LIN {X -30.144,Y 21.431,Z -152.349,A 90.000,B 90.000,C 0.000} C_DIS
LIN {X -28.451,Y 21.431,Z -154.021,A 90.000,B 90.000,C 0.000} C_DIS
LIN {X -26.721,Y 21.431,Z -155.654,A 90.000,B 90.000,C 0.000} C_DIS
LIN {X -24.954,Y 21.431,Z -157.248,A 90.000,B 90.000,C 0.000} C_DIS
LIN {X -23.391,Y 21.431,Z -158.620,A 90.000,B 90.000,C 0.000} C_DIS
LIN {X -21.866,Y 21.431,Z -160.034,A 90.000,B 90.000,C 0.000} C_DIS
LIN {X -20.381,Y 21.431,Z -161.489,A 90.000,B 90.000,C 0.000} C_DIS
LIN {X -18.936,Y 21.431,Z -162.985,A 90.000,B 90.000,C 0.000} C_DIS
LIN {X -18.816,Y 21.431,Z -163.139,A 90.000,B 90.000,C 0.000} C_DIS
LIN {X -18.465,Y 21.431,Z -163.537,A 90.000,B 90.000,C 0.000} C_DIS
LIN {X -18.745,Y 21.431,Z -164.193,A 90.000,B 90.000,C 0.000} C_DIS
LIN {X -19.053,Y 21.431,Z -164.837,A 90.000,B 90.000,C 0.000} C_DIS
LIN {X -19.388,Y 21.431,Z -165.467,A 90.000,B 90.000,C 0.000} C_DIS
LIN {X -20.384,Y 21.431,Z -167.015,A 90.000,B 90.000,C 0.000} C_DIS
LIN {X -21.432,Y 21.431,Z -168.529,A 90.000,B 90.000,C 0.000} C_DIS
LIN {X -22.530,Y 21.431,Z -170.007,A 90.000,B 90.000,C 0.000} C_DIS
LIN {X -23.679,Y 21.431,Z -171.446,A 90.000,B 90.000,C 0.000} C_DIS
LIN {X -24.875,Y 21.431,Z -172.845,A 90.000,B 90.000,C 0.000} C_DIS
LIN {X -26.119,Y 21.431,Z -174.203,A 90.000,B 90.000,C 0.000} C_DIS
LIN {X -27.407,Y 21.431,Z -175.517,A 90.000,B 90.000,C 0.000} C_DIS
LIN {X -28.740,Y 21.431,Z -176.788,A 90.000,B 90.000,C 0.000} C_DIS
LIN {X -30.115,Y 21.431,Z -178.012,A 90.000,B 90.000,C 0.000} C_DIS
LIN {X -33.824,Y 21.431,Z -181.091,A 90.000,B 90.000,C 0.000} C_DIS
LIN {X -37.575,Y 21.431,Z -184.119,A 90.000,B 90.000,C 0.000} C_DIS
LIN {X -41.368,Y 21.431,Z -187.094,A 90.000,B 90.000,C 0.000} C_DIS
LIN {X -45.202,Y 21.431,Z -190.016,A 90.000,B 90.000,C 0.000} C_DIS
LIN {X -49.076,Y 21.431,Z -192.884,A 90.000,B 90.000,C 0.000} C_DIS
LIN {X -52.990,Y 21.431,Z -195.698,A 90.000,B 90.000,C 0.000} C_DIS
LIN {X -56.942,Y 21.431,Z -198.458,A 90.000,B 90.000,C 0.000} C_DIS
LIN {X -60.933,Y 21.431,Z -201.162,A 90.000,B 90.000,C 0.000} C_DIS
LIN {X -64.961,Y 21.431,Z -203.810,A 90.000,B 90.000,C 0.000} C_DIS
LIN {X -71.435,Y 21.431,Z -208.001,A 90.000,B 90.000,C 0.000} C_DIS
LIN {X -77.876,Y 21.431,Z -212.245,A 90.000,B 90.000,C 0.000} C_DIS
LIN {X -84.282,Y 21.431,Z -216.541,A 90.000,B 90.000,C 0.000} C_DIS
LIN {X -90.653,Y 21.431,Z -220.888,A 90.000,B 90.000,C 0.000} C_DIS
LIN {X -96.988,Y 21.431,Z -225.287,A 90.000,B 90.000,C 0.000} C_DIS
LIN {X -101.728,Y 21.431,Z -228.575,A 90.000,B 90.000,C 0.000} C_DIS
LIN {X -107.096,Y 21.431,Z -232.379,A 90.000,B 90.000,C 0.000} C_DIS
LIN {X -112.491,Y 21.431,Z -236.145,A 90.000,B 90.000,C 0.000} C_DIS
LIN {X -117.912,Y 21.431,Z -239.872,A 90.000,B 90.000,C 0.000} C_DIS
LIN {X -123.359,Y 21.431,Z -243.561,A 90.000,B 90.000,C 0.000} C_DIS
LIN {X -145.015,Y 21.431,Z -243.561,A 90.000,B 90.000,C 0.000} C_DIS
LIN {X -145.015,Y 21.431,Z 0.000,A 90.000,B 90.000,C 0.000} C_DIS
LIN {X -145.015,Y 33.931,Z 0.000,A 90.000,B 90.000,C 0.000} C_DIS
LIN {X -145.015,Y 46.431,Z 0.000,A 90.000,B 90.000,C 0.000} C_DIS
LIN {X -145.015,Y 55.062,Z 0.000,A 90.000,B 90.000,C 0.000} C_DIS
LIN {X 100.302,Y 55.062,Z -242.561,A 90.000,B 90.000,C 0.000} C_DIS
LIN {X 100.302,Y 39.288,Z -242.561,A 90.000,B 90.000,C 0.000} C_DIS
LIN {X 100.302,Y 26.788,Z -242.561,A 90.000,B 90.000,C 0.000} C_DIS
LIN {X 100.302,Y 14.287,Z -242.561,A 90.000,B 90.000,C 0.000} C_DIS
LIN {X 144.015,Y 14.287,Z -242.561,A 90.000,B 90.000,C 0.000} C_DIS
LIN {X 144.015,Y 14.287,Z -235.012,A 90.000,B 90.000,C 0.000} C_DIS
LIN {X 102.620,Y 14.287,Z -235.012,A 90.000,B 90.000,C 0.000} C_DIS
LIN {X 103.410,Y 14.287,Z -232.279,A 90.000,B 90.000,C 0.000} C_DIS
LIN {X 104.175,Y 14.287,Z -229.540,A 90.000,B 90.000,C 0.000} C_DIS
LIN {X 104.688,Y 14.287,Z -227.464,A 90.000,B 90.000,C 0.000} C_DIS
LIN {X 144.015,Y 14.287,Z -227.464,A 90.000,B 90.000,C 0.000} C_DIS
LIN {X 144.015,Y 14.287,Z -219.915,A 90.000,B 90.000,C 0.000} C_DIS
LIN {X 106.467,Y 14.287,Z -219.915,A 90.000,B 90.000,C 0.000} C_DIS
LIN {X 107.307,Y 14.287,Z -216.144,A 90.000,B 90.000,C 0.000} C_DIS
LIN {X 108.116,Y 14.287,Z -212.366,A 90.000,B 90.000,C 0.000} C_DIS
LIN {X 144.015,Y 14.287,Z -212.366,A 90.000,B 90.000,C 0.000} C_DIS
LIN {X 144.015,Y 14.287,Z -204.817,A 90.000,B 90.000,C 0.000} C_DIS
LIN {X 109.635,Y 14.287,Z -204.817,A 90.000,B 90.000,C 0.000} C_DIS
LIN {X 110.346,Y 14.287,Z -201.046,A 90.000,B 90.000,C 0.000} C_DIS
LIN {X 111.025,Y 14.287,Z -197.269,A 90.000,B 90.000,C 0.000} C_DIS
LIN {X 144.015,Y 14.287,Z -197.269,A 90.000,B 90.000,C 0.000} C_DIS
LIN {X 144.015,Y 14.287,Z -189.720,A 90.000,B 90.000,C 0.000} C_DIS
LIN {X 112.289,Y 14.287,Z -189.720,A 90.000,B 90.000,C 0.000} C_DIS
LIN {X 112.873,Y 14.287,Z -185.948,A 90.000,B 90.000,C 0.000} C_DIS
LIN {X 113.426,Y 14.287,Z -182.171,A 90.000,B 90.000,C 0.000} C_DIS
LIN {X 144.015,Y 14.287,Z -182.171,A 90.000,B 90.000,C 0.000} C_DIS
LIN {X 144.015,Y 14.287,Z -174.622,A 90.000,B 90.000,C 0.000} C_DIS
LIN {X 114.438,Y 14.287,Z -174.622,A 90.000,B 90.000,C 0.000} C_DIS
LIN {X 114.897,Y 14.287,Z -170.849,A 90.000,B 90.000,C 0.000} C_DIS
LIN {X 115.326,Y 14.287,Z -167.073,A 90.000,B 90.000,C 0.000} C_DIS
LIN {X 144.015,Y 14.287,Z -167.073,A 90.000,B 90.000,C 0.000} C_DIS
LIN {X 144.015,Y 14.287,Z -159.525,A 90.000,B 90.000,C 0.000} C_DIS
LIN {X 116.227,Y 14.287,Z -159.525,A 90.000,B 90.000,C 0.000} C_DIS
LIN {X 116.473,Y 14.287,Z -157.011,A 90.000,B 90.000,C 0.000} C_DIS
LIN {X 116.688,Y 14.287,Z -154.495,A 90.000,B 90.000,C 0.000} C_DIS
LIN {X 116.873,Y 14.287,Z -151.976,A 90.000,B 90.000,C 0.000} C_DIS
LIN {X 144.015,Y 14.287,Z -151.976,A 90.000,B 90.000,C 0.000} C_DIS
LIN {X 144.015,Y 14.287,Z -144.427,A 90.000,B 90.000,C 0.000} C_DIS
LIN {X 117.247,Y 14.287,Z -144.427,A 90.000,B 90.000,C 0.000} C_DIS
LIN {X 117.311,Y 14.287,Z -141.911,A 90.000,B 90.000,C 0.000} C_DIS
LIN {X 117.346,Y 14.287,Z -139.395,A 90.000,B 90.000,C 0.000} C_DIS
LIN {X 117.350,Y 14.287,Z -136.878,A 90.000,B 90.000,C 0.000} C_DIS
LIN {X 144.015,Y 14.287,Z -136.878,A 90.000,B 90.000,C 0.000} C_DIS
LIN {X 144.015,Y 14.287,Z -129.329,A 90.000,B 90.000,C 0.000} C_DIS
LIN {X 117.183,Y 14.287,Z -129.329,A 90.000,B 90.000,C 0.000} C_DIS
LIN {X 117.163,Y 14.287,Z -128.828,A 90.000,B 90.000,C 0.000} C_DIS
LIN {X 117.003,Y 14.287,Z -126.477,A 90.000,B 90.000,C 0.000} C_DIS
LIN {X 116.820,Y 14.287,Z -124.128,A 90.000,B 90.000,C 0.000} C_DIS
LIN {X 116.613,Y 14.287,Z -121.781,A 90.000,B 90.000,C 0.000} C_DIS
LIN {X 144.015,Y 14.287,Z -121.781,A 90.000,B 90.000,C 0.000} C_DIS
LIN {X 144.015,Y 14.287,Z -114.232,A 90.000,B 90.000,C 0.000} C_DIS
LIN {X 115.786,Y 14.287,Z -114.232,A 90.000,B 90.000,C 0.000} C_DIS
LIN {X 115.455,Y 14.287,Z -111.712,A 90.000,B 90.000,C 0.000} C_DIS
LIN {X 115.097,Y 14.287,Z -109.195,A 90.000,B 90.000,C 0.000} C_DIS
LIN {X 114.712,Y 14.287,Z -106.683,A 90.000,B 90.000,C 0.000} C_DIS
LIN {X 144.015,Y 14.287,Z -106.683,A 90.000,B 90.000,C 0.000} C_DIS
LIN {X 144.015,Y 14.287,Z -99.134,A 90.000,B 90.000,C 0.000} C_DIS
LIN {X 113.387,Y 14.287,Z -99.134,A 90.000,B 90.000,C 0.000} C_DIS
LIN {X 113.108,Y 14.287,Z -97.708,A 90.000,B 90.000,C 0.000} C_DIS
LIN {X 112.820,Y 14.287,Z -96.283,A 90.000,B 90.000,C 0.000} C_DIS
LIN {X 112.622,Y 14.287,Z -95.095,A 90.000,B 90.000,C 0.000} C_DIS
LIN {X 112.380,Y 14.287,Z -93.915,A 90.000,B 90.000,C 0.000} C_DIS
LIN {X 112.094,Y 14.287,Z -92.745,A 90.000,B 90.000,C 0.000} C_DIS
LIN {X 111.765,Y 14.287,Z -91.586,A 90.000,B 90.000,C 0.000} C_DIS
LIN {X 144.015,Y 14.287,Z -91.586,A 90.000,B 90.000,C 0.000} C_DIS
LIN {X 144.015,Y 14.287,Z -84.037,A 90.000,B 90.000,C 0.000} C_DIS
LIN {X 110.092,Y 14.287,Z -84.037,A 90.000,B 90.000,C 0.000} C_DIS
LIN {X 111.141,Y 14.287,Z -82.191,A 90.000,B 90.000,C 0.000} C_DIS
LIN {X 112.138,Y 14.287,Z -80.316,A 90.000,B 90.000,C 0.000} C_DIS
LIN {X 113.084,Y 14.287,Z -78.415,A 90.000,B 90.000,C 0.000} C_DIS
LIN {X 113.977,Y 14.287,Z -76.488,A 90.000,B 90.000,C 0.000} C_DIS
LIN {X 144.015,Y 14.287,Z -76.488,A 90.000,B 90.000,C 0.000} C_DIS
LIN {X 144.015,Y 14.287,Z -68.939,A 90.000,B 90.000,C 0.000} C_DIS
LIN {X 116.890,Y 14.287,Z -68.939,A 90.000,B 90.000,C 0.000} C_DIS
LIN {X 117.231,Y 14.287,Z -67.869,A 90.000,B 90.000,C 0.000} C_DIS
LIN {X 117.556,Y 14.287,Z -66.794,A 90.000,B 90.000,C 0.000} C_DIS
LIN {X 118.300,Y 14.287,Z -64.088,A 90.000,B 90.000,C 0.000} C_DIS
LIN {X 119.069,Y 14.287,Z -61.390,A 90.000,B 90.000,C 0.000} C_DIS
LIN {X 144.015,Y 14.287,Z -61.390,A 90.000,B 90.000,C 0.000} C_DIS
LIN {X 144.015,Y 14.287,Z -53.842,A 90.000,B 90.000,C 0.000} C_DIS
LIN {X 122.274,Y 14.287,Z -53.842,A 90.000,B 90.000,C 0.000} C_DIS
LIN {X 122.630,Y 14.287,Z -53.139,A 90.000,B 90.000,C 0.000} C_DIS
LIN {X 122.993,Y 14.287,Z -52.439,A 90.000,B 90.000,C 0.000} C_DIS
LIN {X 123.486,Y 14.287,Z -51.468,A 90.000,B 90.000,C 0.000} C_DIS
LIN {X 123.926,Y 14.287,Z -50.472,A 90.000,B 90.000,C 0.000} C_DIS
LIN {X 124.312,Y 14.287,Z -49.453,A 90.000,B 90.000,C 0.000} C_DIS
LIN {X 124.641,Y 14.287,Z -48.415,A 90.000,B 90.000,C 0.000} C_DIS
LIN {X 124.915,Y 14.287,Z -47.360,A 90.000,B 90.000,C 0.000} C_DIS
LIN {X 125.131,Y 14.287,Z -46.293,A 90.000,B 90.000,C 0.000} C_DIS
LIN {X 144.015,Y 14.287,Z -46.293,A 90.000,B 90.000,C 0.000} C_DIS
LIN {X 144.015,Y 14.287,Z -38.744,A 90.000,B 90.000,C 0.000} C_DIS
LIN {X 125.030,Y 14.287,Z -38.744,A 90.000,B 90.000,C 0.000} C_DIS
LIN {X 124.784,Y 14.287,Z -37.789,A 90.000,B 90.000,C 0.000} C_DIS
LIN {X 124.472,Y 14.287,Z -36.853,A 90.000,B 90.000,C 0.000} C_DIS
LIN {X 124.097,Y 14.287,Z -35.940,A 90.000,B 90.000,C 0.000} C_DIS
LIN {X 123.660,Y 14.287,Z -35.056,A 90.000,B 90.000,C 0.000} C_DIS
LIN {X 123.164,Y 14.287,Z -34.204,A 90.000,B 90.000,C 0.000} C_DIS
LIN {X 122.609,Y 14.287,Z -33.388,A 90.000,B 90.000,C 0.000} C_DIS
LIN {X 122.000,Y 14.287,Z -32.612,A 90.000,B 90.000,C 0.000} C_DIS
LIN {X 121.339,Y 14.287,Z -31.880,A 90.000,B 90.000,C 0.000} C_DIS
LIN {X 120.629,Y 14.287,Z -31.195,A 90.000,B 90.000,C 0.000} C_DIS
LIN {X 144.015,Y 14.287,Z -31.195,A 90.000,B 90.000,C 0.000} C_DIS
LIN {X 144.015,Y 14.287,Z -23.646,A 90.000,B 90.000,C 0.000} C_DIS
LIN {X 5.340,Y 14.287,Z -23.646,A 90.000,B 90.000,C 0.000} C_DIS
LIN {X 2.315,Y 14.287,Z -23.147,A 90.000,B 90.000,C 0.000} C_DIS
LIN {X -0.703,Y 14.287,Z -22.607,A 90.000,B 90.000,C 0.000} C_DIS
LIN {X -3.714,Y 14.287,Z -22.027,A 90.000,B 90.000,C 0.000} C_DIS
LIN {X -6.716,Y 14.287,Z -21.406,A 90.000,B 90.000,C 0.000} C_DIS
LIN {X -9.710,Y 14.287,Z -20.745,A 90.000,B 90.000,C 0.000} C_DIS
LIN {X -13.667,Y 14.287,Z -19.813,A 90.000,B 90.000,C 0.000} C_DIS
LIN {X -17.634,Y 14.287,Z -18.928,A 90.000,B 90.000,C 0.000} C_DIS
LIN {X -21.612,Y 14.287,Z -18.088,A 90.000,B 90.000,C 0.000} C_DIS
LIN {X -25.599,Y 14.287,Z -17.295,A 90.000,B 90.000,C 0.000} C_DIS
LIN {X -27.541,Y 14.287,Z -16.862,A 90.000,B 90.000,C 0.000} C_DIS
LIN {X -29.491,Y 14.287,Z -16.463,A 90.000,B 90.000,C 0.000} C_DIS
LIN {X -31.447,Y 14.287,Z -16.098,A 90.000,B 90.000,C 0.000} C_DIS
LIN {X 144.015,Y 14.287,Z -16.098,A 90.000,B 90.000,C 0.000} C_DIS
LIN {X 144.015,Y 14.287,Z -8.549,A 90.000,B 90.000,C 0.000} C_DIS
LIN {X -67.014,Y 14.287,Z -8.549,A 90.000,B 90.000,C 0.000} C_DIS
LIN {X -68.321,Y 14.287,Z -7.964,A 90.000,B 90.000,C 0.000} C_DIS
LIN {X -69.464,Y 14.287,Z -7.415,A 90.000,B 90.000,C 0.000} C_DIS
LIN {X -70.635,Y 14.287,Z -6.927,A 90.000,B 90.000,C 0.000} C_DIS
LIN {X -71.829,Y 14.287,Z -6.502,A 90.000,B 90.000,C 0.000} C_DIS
LIN {X -73.045,Y 14.287,Z -6.142,A 90.000,B 90.000,C 0.000} C_DIS
LIN {X -74.279,Y 14.287,Z -5.847,A 90.000,B 90.000,C 0.000} C_DIS
LIN {X -75.526,Y 14.287,Z -5.618,A 90.000,B 90.000,C 0.000} C_DIS
LIN {X -76.784,Y 14.287,Z -5.456,A 90.000,B 90.000,C 0.000} C_DIS
LIN {X -78.048,Y 14.287,Z -5.361,A 90.000,B 90.000,C 0.000} C_DIS
LIN {X -79.316,Y 14.287,Z -5.334,A 90.000,B 90.000,C 0.000} C_DIS
LIN {X -80.584,Y 14.287,Z -5.375,A 90.000,B 90.000,C 0.000} C_DIS
LIN {X -81.847,Y 14.287,Z -5.483,A 90.000,B 90.000,C 0.000} C_DIS
LIN {X -83.103,Y 14.287,Z -5.658,A 90.000,B 90.000,C 0.000} C_DIS
LIN {X -84.348,Y 14.287,Z -5.899,A 90.000,B 90.000,C 0.000} C_DIS
LIN {X -85.303,Y 14.287,Z -6.093,A 90.000,B 90.000,C 0.000} C_DIS
LIN {X -86.243,Y 14.287,Z -6.351,A 90.000,B 90.000,C 0.000} C_DIS
LIN {X -87.163,Y 14.287,Z -6.671,A 90.000,B 90.000,C 0.000} C_DIS
LIN {X -88.060,Y 14.287,Z -7.052,A 90.000,B 90.000,C 0.000} C_DIS
LIN {X -88.929,Y 14.287,Z -7.492,A 90.000,B 90.000,C 0.000} C_DIS
LIN {X -89.767,Y 14.287,Z -7.990,A 90.000,B 90.000,C 0.000} C_DIS
LIN {X -90.843,Y 14.287,Z -8.053,A 90.000,B 90.000,C 0.000} C_DIS
LIN {X -91.915,Y 14.287,Z -8.167,A 90.000,B 90.000,C 0.000} C_DIS
LIN {X -92.981,Y 14.287,Z -8.332,A 90.000,B 90.000,C 0.000} C_DIS
LIN {X -94.037,Y 14.287,Z -8.549,A 90.000,B 90.000,C 0.000} C_DIS
LIN {X -144.015,Y 14.287,Z -8.549,A 90.000,B 90.000,C 0.000} C_DIS
LIN {X -144.015,Y 14.287,Z -16.098,A 90.000,B 90.000,C 0.000} C_DIS
LIN {X -106.655,Y 14.287,Z -16.098,A 90.000,B 90.000,C 0.000} C_DIS
LIN {X -107.024,Y 14.287,Z -16.531,A 90.000,B 90.000,C 0.000} C_DIS
LIN {X -107.373,Y 14.287,Z -16.981,A 90.000,B 90.000,C 0.000} C_DIS
LIN {X -108.462,Y 14.287,Z -17.322,A 90.000,B 90.000,C 0.000} C_DIS
LIN {X -109.531,Y 14.287,Z -17.720,A 90.000,B 90.000,C 0.000} C_DIS
LIN {X -110.578,Y 14.287,Z -18.174,A 90.000,B 90.000,C 0.000} C_DIS
LIN {X -111.598,Y 14.287,Z -18.684,A 90.000,B 90.000,C 0.000} C_DIS
LIN {X -112.591,Y 14.287,Z -19.246,A 90.000,B 90.000,C 0.000} C_DIS
LIN {X -113.552,Y 14.287,Z -19.861,A 90.000,B 90.000,C 0.000} C_DIS
LIN {X -114.479,Y 14.287,Z -20.526,A 90.000,B 90.000,C 0.000} C_DIS
LIN {X -115.370,Y 14.287,Z -21.239,A 90.000,B 90.000,C 0.000} C_DIS
LIN {X -116.222,Y 14.287,Z -21.998,A 90.000,B 90.000,C 0.000} C_DIS
LIN {X -117.032,Y 14.287,Z -22.801,A 90.000,B 90.000,C 0.000} C_DIS
LIN {X -117.799,Y 14.287,Z -23.646,A 90.000,B 90.000,C 0.000} C_DIS
LIN {X -144.015,Y 14.287,Z -23.646,A 90.000,B 90.000,C 0.000} C_DIS
LIN {X -144.015,Y 14.287,Z -31.195,A 90.000,B 90.000,C 0.000} C_DIS
LIN {X -122.817,Y 14.287,Z -31.195,A 90.000,B 90.000,C 0.000} C_DIS
LIN {X -123.177,Y 14.287,Z -32.233,A 90.000,B 90.000,C 0.000} C_DIS
LIN {X -123.472,Y 14.287,Z -33.291,A 90.000,B 90.000,C 0.000} C_DIS
LIN {X -123.701,Y 14.287,Z -34.366,A 90.000,B 90.000,C 0.000} C_DIS
LIN {X -123.861,Y 14.287,Z -35.453,A 90.000,B 90.000,C 0.000} C_DIS
LIN {X -123.954,Y 14.287,Z -36.548,A 90.000,B 90.000,C 0.000} C_DIS
LIN {X -123.979,Y 14.287,Z -37.646,A 90.000,B 90.000,C 0.000} C_DIS
LIN {X -123.934,Y 14.287,Z -38.744,A 90.000,B 90.000,C 0.000} C_DIS
LIN {X -144.015,Y 14.287,Z -38.744,A 90.000,B 90.000,C 0.000} C_DIS
LIN {X -144.015,Y 14.287,Z -46.293,A 90.000,B 90.000,C 0.000} C_DIS
LIN {X -123.207,Y 14.287,Z -46.293,A 90.000,B 90.000,C 0.000} C_DIS
LIN {X -123.190,Y 14.287,Z -47.313,A 90.000,B 90.000,C 0.000} C_DIS
LIN {X -123.108,Y 14.287,Z -48.329,A 90.000,B 90.000,C 0.000} C_DIS
LIN {X -122.962,Y 14.287,Z -49.339,A 90.000,B 90.000,C 0.000} C_DIS
LIN {X -122.752,Y 14.287,Z -50.337,A 90.000,B 90.000,C 0.000} C_DIS
LIN {X -122.479,Y 14.287,Z -51.320,A 90.000,B 90.000,C 0.000} C_DIS
LIN {X -122.144,Y 14.287,Z -52.283,A 90.000,B 90.000,C 0.000} C_DIS
LIN {X -121.748,Y 14.287,Z -53.223,A 90.000,B 90.000,C 0.000} C_DIS
LIN {X -121.595,Y 14.287,Z -53.842,A 90.000,B 90.000,C 0.000} C_DIS
LIN {X -144.015,Y 14.287,Z -53.842,A 90.000,B 90.000,C 0.000} C_DIS
LIN {X -144.015,Y 14.287,Z -61.390,A 90.000,B 90.000,C 0.000} C_DIS
LIN {X -119.537,Y 14.287,Z -61.390,A 90.000,B 90.000,C 0.000} C_DIS
LIN {X -119.056,Y 14.287,Z -62.708,A 90.000,B 90.000,C 0.000} C_DIS
LIN {X -118.522,Y 14.287,Z -64.005,A 90.000,B 90.000,C 0.000} C_DIS
LIN {X -117.934,Y 14.287,Z -65.279,A 90.000,B 90.000,C 0.000} C_DIS
LIN {X -117.295,Y 14.287,Z -66.527,A 90.000,B 90.000,C 0.000} C_DIS
LIN {X -116.604,Y 14.287,Z -67.748,A 90.000,B 90.000,C 0.000} C_DIS
LIN {X -115.863,Y 14.287,Z -68.939,A 90.000,B 90.000,C 0.000} C_DIS
LIN {X -144.015,Y 14.287,Z -68.939,A 90.000,B 90.000,C 0.000} C_DIS
LIN {X -144.015,Y 14.287,Z -76.488,A 90.000,B 90.000,C 0.000} C_DIS
LIN {X -109.288,Y 14.287,Z -76.488,A 90.000,B 90.000,C 0.000} C_DIS
LIN {X -108.521,Y 14.287,Z -77.148,A 90.000,B 90.000,C 0.000} C_DIS
LIN {X -107.719,Y 14.287,Z -77.766,A 90.000,B 90.000,C 0.000} C_DIS
LIN {X -106.886,Y 14.287,Z -78.340,A 90.000,B 90.000,C 0.000} C_DIS
LIN {X -106.023,Y 14.287,Z -78.868,A 90.000,B 90.000,C 0.000} C_DIS
LIN {X -105.133,Y 14.287,Z -79.350,A 90.000,B 90.000,C 0.000} C_DIS
LIN {X -104.218,Y 14.287,Z -79.783,A 90.000,B 90.000,C 0.000} C_DIS
LIN {X -104.128,Y 14.287,Z -79.831,A 90.000,B 90.000,C 0.000} C_DIS
LIN {X -103.286,Y 14.287,Z -80.260,A 90.000,B 90.000,C 0.000} C_DIS
LIN {X -102.420,Y 14.287,Z -80.639,A 90.000,B 90.000,C 0.000} C_DIS
LIN {X -101.534,Y 14.287,Z -80.966,A 90.000,B 90.000,C 0.000} C_DIS
LIN {X -100.630,Y 14.287,Z -81.241,A 90.000,B 90.000,C 0.000} C_DIS
LIN {X -99.711,Y 14.287,Z -81.461,A 90.000,B 90.000,C 0.000} C_DIS
LIN {X -98.781,Y 14.287,Z -81.628,A 90.000,B 90.000,C 0.000} C_DIS
LIN {X -98.628,Y 14.287,Z -81.664,A 90.000,B 90.000,C 0.000} C_DIS
LIN {X -96.905,Y 14.287,Z -81.904,A 90.000,B 90.000,C 0.000} C_DIS
LIN {X -95.177,Y 14.287,Z -82.109,A 90.000,B 90.000,C 0.000} C_DIS
LIN {X -93.445,Y 14.287,Z -82.279,A 90.000,B 90.000,C 0.000} C_DIS
LIN {X -93.383,Y 14.287,Z -82.289,A 90.000,B 90.000,C 0.000} C_DIS
LIN {X -92.938,Y 14.287,Z -82.457,A 90.000,B 90.000,C 0.000} C_DIS
LIN {X -92.507,Y 14.287,Z -82.659,A 90.000,B 90.000,C 0.000} C_DIS
LIN {X -92.093,Y 14.287,Z -82.893,A 90.000,B 90.000,C 0.000} C_DIS
LIN {X -91.698,Y 14.287,Z -83.159,A 90.000,B 90.000,C 0.000} C_DIS
LIN {X -91.216,Y 14.287,Z -83.601,A 90.000,B 90.000,C 0.000} C_DIS
LIN {X -90.729,Y 14.287,Z -84.037,A 90.000,B 90.000,C 0.000} C_DIS
LIN {X -144.015,Y 14.287,Z -84.037,A 90.000,B 90.000,C 0.000} C_DIS
LIN {X -144.015,Y 14.287,Z -91.586,A 90.000,B 90.000,C 0.000} C_DIS
LIN {X -80.184,Y 14.287,Z -91.586,A 90.000,B 90.000,C 0.000} C_DIS
LIN {X -78.153,Y 14.287,Z -92.888,A 90.000,B 90.000,C 0.000} C_DIS
LIN {X -76.910,Y 14.287,Z -93.660,A 90.000,B 90.000,C 0.000} C_DIS
LIN {X -75.693,Y 14.287,Z -94.474,A 90.000,B 90.000,C 0.000} C_DIS
LIN {X -74.505,Y 14.287,Z -95.329,A 90.000,B 90.000,C 0.000} C_DIS
LIN {X -73.346,Y 14.287,Z -96.223,A 90.000,B 90.000,C 0.000} C_DIS
LIN {X -72.219,Y 14.287,Z -97.156,A 90.000,B 90.000,C 0.000} C_DIS
LIN {X -71.123,Y 14.287,Z -98.127,A 90.000,B 90.000,C 0.000} C_DIS
LIN {X -70.061,Y 14.287,Z -99.134,A 90.000,B 90.000,C 0.000} C_DIS
LIN {X -144.015,Y 14.287,Z -99.134,A 90.000,B 90.000,C 0.000} C_DIS
LIN {X -144.015,Y 14.287,Z -106.683,A 90.000,B 90.000,C 0.000} C_DIS
LIN {X -63.845,Y 14.287,Z -106.683,A 90.000,B 90.000,C 0.000} C_DIS
LIN {X -61.945,Y 14.287,Z -109.223,A 90.000,B 90.000,C 0.000} C_DIS
LIN {X -60.014,Y 14.287,Z -111.739,A 90.000,B 90.000,C 0.000} C_DIS
LIN {X -58.052,Y 14.287,Z -114.232,A 90.000,B 90.000,C 0.000} C_DIS
LIN {X -144.015,Y 14.287,Z -114.232,A 90.000,B 90.000,C 0.000} C_DIS
LIN {X -144.015,Y 14.287,Z -121.781,A 90.000,B 90.000,C 0.000} C_DIS
LIN {X -51.816,Y 14.287,Z -121.781,A 90.000,B 90.000,C 0.000} C_DIS
LIN {X -50.808,Y 14.287,Z -123.147,A 90.000,B 90.000,C 0.000} C_DIS
LIN {X -49.834,Y 14.287,Z -124.538,A 90.000,B 90.000,C 0.000} C_DIS
LIN {X -49.055,Y 14.287,Z -126.117,A 90.000,B 90.000,C 0.000} C_DIS
LIN {X -48.313,Y 14.287,Z -127.715,A 90.000,B 90.000,C 0.000} C_DIS
LIN {X -47.609,Y 14.287,Z -129.329,A 90.000,B 90.000,C 0.000} C_DIS
LIN {X -144.015,Y 14.287,Z -129.329,A 90.000,B 90.000,C 0.000} C_DIS
LIN {X -144.015,Y 14.287,Z -136.878,A 90.000,B 90.000,C 0.000} C_DIS
LIN {X -44.292,Y 14.287,Z -136.878,A 90.000,B 90.000,C 0.000} C_DIS
LIN {X -43.485,Y 14.287,Z -138.431,A 90.000,B 90.000,C 0.000} C_DIS
LIN {X -42.639,Y 14.287,Z -139.963,A 90.000,B 90.000,C 0.000} C_DIS
LIN {X -41.756,Y 14.287,Z -141.473,A 90.000,B 90.000,C 0.000} C_DIS
LIN {X -40.836,Y 14.287,Z -142.962,A 90.000,B 90.000,C 0.000} C_DIS
LIN {X -39.879,Y 14.287,Z -144.427,A 90.000,B 90.000,C 0.000} C_DIS
LIN {X -144.015,Y 14.287,Z -144.427,A 90.000,B 90.000,C 0.000} C_DIS
LIN {X -144.015,Y 14.287,Z -151.976,A 90.000,B 90.000,C 0.000} C_DIS
LIN {X -33.972,Y 14.287,Z -151.976,A 90.000,B 90.000,C 0.000} C_DIS
LIN {X -31.573,Y 14.287,Z -154.527,A 90.000,B 90.000,C 0.000} C_DIS
LIN {X -29.138,Y 14.287,Z -157.044,A 90.000,B 90.000,C 0.000} C_DIS
LIN {X -26.667,Y 14.287,Z -159.525,A 90.000,B 90.000,C 0.000} C_DIS
LIN {X -144.015,Y 14.287,Z -159.525,A 90.000,B 90.000,C 0.000} C_DIS
LIN {X -144.015,Y 14.287,Z -167.073,A 90.000,B 90.000,C 0.000} C_DIS
LIN {X -26.448,Y 14.287,Z -167.073,A 90.000,B 90.000,C 0.000} C_DIS
LIN {X -27.323,Y 14.287,Z -168.257,A 90.000,B 90.000,C 0.000} C_DIS
LIN {X -28.242,Y 14.287,Z -169.409,A 90.000,B 90.000,C 0.000} C_DIS
LIN {X -29.201,Y 14.287,Z -170.526,A 90.000,B 90.000,C 0.000} C_DIS
LIN {X -30.201,Y 14.287,Z -171.607,A 90.000,B 90.000,C 0.000} C_DIS
LIN {X -31.239,Y 14.287,Z -172.651,A 90.000,B 90.000,C 0.000} C_DIS
LIN {X -32.315,Y 14.287,Z -173.657,A 90.000,B 90.000,C 0.000} C_DIS
LIN {X -33.427,Y 14.287,Z -174.622,A 90.000,B 90.000,C 0.000} C_DIS
LIN {X -144.015,Y 14.287,Z -174.622,A 90.000,B 90.000,C 0.000} C_DIS
LIN {X -144.015,Y 14.287,Z -182.171,A 90.000,B 90.000,C 0.000} C_DIS
LIN {X -43.393,Y 14.287,Z -182.171,A 90.000,B 90.000,C 0.000} C_DIS
LIN {X -46.143,Y 14.287,Z -184.116,A 90.000,B 90.000,C 0.000} C_DIS
LIN {X -48.919,Y 14.287,Z -186.023,A 90.000,B 90.000,C 0.000} C_DIS
LIN {X -51.722,Y 14.287,Z -187.891,A 90.000,B 90.000,C 0.000} C_DIS
LIN {X -54.550,Y 14.287,Z -189.720,A 90.000,B 90.000,C 0.000} C_DIS
LIN {X -144.015,Y 14.287,Z -189.720,A 90.000,B 90.000,C 0.000} C_DIS
LIN {X -144.015,Y 14.287,Z -197.269,A 90.000,B 90.000,C 0.000} C_DIS
LIN {X -66.947,Y 14.287,Z -197.269,A 90.000,B 90.000,C 0.000} C_DIS
LIN {X -71.176,Y 14.287,Z -199.763,A 90.000,B 90.000,C 0.000} C_DIS
LIN {X -75.391,Y 14.287,Z -202.279,A 90.000,B 90.000,C 0.000} C_DIS
LIN {X -79.594,Y 14.287,Z -204.817,A 90.000,B 90.000,C 0.000} C_DIS
LIN {X -144.015,Y 14.287,Z -204.817,A 90.000,B 90.000,C 0.000} C_DIS
LIN {X -144.015,Y 14.287,Z -212.366,A 90.000,B 90.000,C 0.000} C_DIS
LIN {X -91.801,Y 14.287,Z -212.366,A 90.000,B 90.000,C 0.000} C_DIS
LIN {X -95.747,Y 14.287,Z -214.862,A 90.000,B 90.000,C 0.000} C_DIS
LIN {X -99.680,Y 14.287,Z -217.379,A 90.000,B 90.000,C 0.000} C_DIS
LIN {X -103.600,Y 14.287,Z -219.915,A 90.000,B 90.000,C 0.000} C_DIS
LIN {X -144.015,Y 14.287,Z -219.915,A 90.000,B 90.000,C 0.000} C_DIS
LIN {X -144.015,Y 14.287,Z -227.464,A 90.000,B 90.000,C 0.000} C_DIS
LIN {X -115.053,Y 14.287,Z -227.464,A 90.000,B 90.000,C 0.000} C_DIS
LIN {X -122.337,Y 14.287,Z -232.351,A 90.000,B 90.000,C 0.000} C_DIS
LIN {X -126.258,Y 14.287,Z -235.012,A 90.000,B 90.000,C 0.000} C_DIS
LIN {X -144.015,Y 14.287,Z -235.012,A 90.000,B 90.000,C 0.000} C_DIS
LIN {X -144.015,Y 14.287,Z -242.561,A 90.000,B 90.000,C 0.000} C_DIS
LIN {X -137.094,Y 14.287,Z -242.561,A 90.000,B 90.000,C 0.000} C_DIS
LIN {X -144.015,Y 14.287,Z -1.000,A 90.000,B 90.000,C 0.000} C_DIS
LIN {X 144.015,Y 14.287,Z -1.000,A 90.000,B 90.000,C 0.000} C_DIS
LIN {X 98.307,Y 14.287,Z -31.195,A 90.000,B 90.000,C 0.000} C_DIS
LIN {X 45.099,Y 14.287,Z -31.195,A 90.000,B 90.000,C 0.000} C_DIS
LIN {X 47.546,Y 14.287,Z -32.059,A 90.000,B 90.000,C 0.000} C_DIS
LIN {X 49.978,Y 14.287,Z -32.965,A 90.000,B 90.000,C 0.000} C_DIS
LIN {X 52.394,Y 14.287,Z -33.911,A 90.000,B 90.000,C 0.000} C_DIS
LIN {X 54.085,Y 14.287,Z -34.773,A 90.000,B 90.000,C 0.000} C_DIS
LIN {X 55.748,Y 14.287,Z -35.689,A 90.000,B 90.000,C 0.000} C_DIS
LIN {X 57.382,Y 14.287,Z -36.656,A 90.000,B 90.000,C 0.000} C_DIS
LIN {X 58.983,Y 14.287,Z -37.675,A 90.000,B 90.000,C 0.000} C_DIS
LIN {X 60.552,Y 14.287,Z -38.744,A 90.000,B 90.000,C 0.000} C_DIS
LIN {X 85.592,Y 14.287,Z -38.744,A 90.000,B 90.000,C 0.000} C_DIS
LIN {X 84.450,Y 14.287,Z -39.711,A 90.000,B 90.000,C 0.000} C_DIS
LIN {X 83.338,Y 14.287,Z -40.714,A 90.000,B 90.000,C 0.000} C_DIS
LIN {X 82.260,Y 14.287,Z -41.752,A 90.000,B 90.000,C 0.000} C_DIS
LIN {X 81.214,Y 14.287,Z -42.823,A 90.000,B 90.000,C 0.000} C_DIS
LIN {X 80.413,Y 14.287,Z -43.639,A 90.000,B 90.000,C 0.000} C_DIS
LIN {X 79.650,Y 14.287,Z -44.490,A 90.000,B 90.000,C 0.000} C_DIS
LIN {X 78.927,Y 14.287,Z -45.375,A 90.000,B 90.000,C 0.000} C_DIS
LIN {X 78.245,Y 14.287,Z -46.293,A 90.000,B 90.000,C 0.000} C_DIS
LIN {X 73.847,Y 14.287,Z -46.293,A 90.000,B 90.000,C 0.000} C_DIS
LIN {X 77.376,Y 14.287,Z -49.619,A 90.000,B 90.000,C 0.000} C_DIS
LIN {X 75.302,Y 14.287,Z -48.325,A 90.000,B 90.000,C 0.000} C_DIS
LIN {X 73.202,Y 14.287,Z -47.074,A 90.000,B 90.000,C 0.000} C_DIS
LIN {X 71.075,Y 14.287,Z -45.869,A 90.000,B 90.000,C 0.000} C_DIS
LIN {X 68.924,Y 14.287,Z -44.709,A 90.000,B 90.000,C 0.000} C_DIS
LIN {X 66.748,Y 14.287,Z -43.594,A 90.000,B 90.000,C 0.000} C_DIS
LIN {X 64.550,Y 14.287,Z -42.525,A 90.000,B 90.000,C 0.000} C_DIS
LIN {X 63.559,Y 14.287,Z -42.002,A 90.000,B 90.000,C 0.000} C_DIS
LIN {X 62.561,Y 14.287,Z -41.493,A 90.000,B 90.000,C 0.000} C_DIS
LIN {X 61.141,Y 14.287,Z -40.405,A 90.000,B 90.000,C 0.000} C_DIS
LIN {X 59.688,Y 14.287,Z -39.360,A 90.000,B 90.000,C 0.000} C_DIS
LIN {X 58.204,Y 14.287,Z -38.361,A 90.000,B 90.000,C 0.000} C_DIS
LIN {X 56.691,Y 14.287,Z -37.406,A 90.000,B 90.000,C 0.000} C_DIS
LIN {X 55.149,Y 14.287,Z -36.498,A 90.000,B 90.000,C 0.000} C_DIS
LIN {X 53.581,Y 14.287,Z -35.638,A 90.000,B 90.000,C 0.000} C_DIS
LIN {X 51.987,Y 14.287,Z -34.825,A 90.000,B 90.000,C 0.000} C_DIS
LIN {X 49.331,Y 14.287,Z -33.789,A 90.000,B 90.000,C 0.000} C_DIS
LIN {X 46.657,Y 14.287,Z -32.802,A 90.000,B 90.000,C 0.000} C_DIS
LIN {X 43.964,Y 14.287,Z -31.865,A 90.000,B 90.000,C 0.000} C_DIS
LIN {X 41.255,Y 14.287,Z -30.978,A 90.000,B 90.000,C 0.000} C_DIS
LIN {X 38.529,Y 14.287,Z -30.142,A 90.000,B 90.000,C 0.000} C_DIS
LIN {X 35.789,Y 14.287,Z -29.356,A 90.000,B 90.000,C 0.000} C_DIS
LIN {X 33.956,Y 14.287,Z -28.833,A 90.000,B 90.000,C 0.000} C_DIS
LIN {X 32.105,Y 14.287,Z -28.373,A 90.000,B 90.000,C 0.000} C_DIS
LIN {X 30.240,Y 14.287,Z -27.976,A 90.000,B 90.000,C 0.000} C_DIS
LIN {X 28.363,Y 14.287,Z -27.644,A 90.000,B 90.000,C 0.000} C_DIS
LIN {X 26.475,Y 14.287,Z -27.375,A 90.000,B 90.000,C 0.000} C_DIS
LIN {X 24.580,Y 14.287,Z -27.172,A 90.000,B 90.000,C 0.000} C_DIS
LIN {X 22.678,Y 14.287,Z -27.034,A 90.000,B 90.000,C 0.000} C_DIS
LIN {X 21.240,Y 14.287,Z -27.123,A 90.000,B 90.000,C 0.000} C_DIS
LIN {X 19.800,Y 14.287,Z -27.159,A 90.000,B 90.000,C 0.000} C_DIS
LIN {X 18.359,Y 14.287,Z -27.141,A 90.000,B 90.000,C 0.000} C_DIS
LIN {X 16.920,Y 14.287,Z -27.069,A 90.000,B 90.000,C 0.000} C_DIS
LIN {X 13.486,Y 14.287,Z -26.291,A 90.000,B 90.000,C 0.000} C_DIS
LIN {X 10.044,Y 14.287,Z -25.553,A 90.000,B 90.000,C 0.000} C_DIS
LIN {X 6.594,Y 14.287,Z -24.852,A 90.000,B 90.000,C 0.000} C_DIS
LIN {X 3.270,Y 14.287,Z -24.323,A 90.000,B 90.000,C 0.000} C_DIS
LIN {X -0.047,Y 14.287,Z -23.745,A 90.000,B 90.000,C 0.000} C_DIS
LIN {X -3.354,Y 14.287,Z -23.118,A 90.000,B 90.000,C 0.000} C_DIS
LIN {X -6.651,Y 14.287,Z -22.442,A 90.000,B 90.000,C 0.000} C_DIS
LIN {X -9.939,Y 14.287,Z -21.719,A 90.000,B 90.000,C 0.000} C_DIS
LIN {X -13.891,Y 14.287,Z -20.789,A 90.000,B 90.000,C 0.000} C_DIS
LIN {X -17.853,Y 14.287,Z -19.904,A 90.000,B 90.000,C 0.000} C_DIS
LIN {X -21.825,Y 14.287,Z -19.066,A 90.000,B 90.000,C 0.000} C_DIS
LIN {X -25.807,Y 14.287,Z -18.274,A 90.000,B 90.000,C 0.000} C_DIS
LIN {X -27.926,Y 14.287,Z -17.803,A 90.000,B 90.000,C 0.000} C_DIS
LIN {X -30.054,Y 14.287,Z -17.373,A 90.000,B 90.000,C 0.000} C_DIS
LIN {X -32.189,Y 14.287,Z -16.983,A 90.000,B 90.000,C 0.000} C_DIS
LIN {X -34.331,Y 14.287,Z -16.634,A 90.000,B 90.000,C 0.000} C_DIS
LIN {X -36.480,Y 14.287,Z -16.326,A 90.000,B 90.000,C 0.000} C_DIS
LIN {X -39.917,Y 14.287,Z -15.920,A 90.000,B 90.000,C 0.000} C_DIS
LIN {X -43.352,Y 14.287,Z -15.497,A 90.000,B 90.000,C 0.000} C_DIS
LIN {X -48.382,Y 14.287,Z -14.794,A 90.000,B 90.000,C 0.000} C_DIS
LIN {X -53.417,Y 14.287,Z -14.125,A 90.000,B 90.000,C 0.000} C_DIS
LIN {X -54.230,Y 14.287,Z -14.089,A 90.000,B 90.000,C 0.000} C_DIS
LIN {X -55.040,Y 14.287,Z -14.011,A 90.000,B 90.000,C 0.000} C_DIS
LIN {X -55.845,Y 14.287,Z -13.891,A 90.000,B 90.000,C 0.000} C_DIS
LIN {X -56.643,Y 14.287,Z -13.730,A 90.000,B 90.000,C 0.000} C_DIS
LIN {X -57.431,Y 14.287,Z -13.528,A 90.000,B 90.000,C 0.000} C_DIS
LIN {X -60.292,Y 14.287,Z -12.436,A 90.000,B 90.000,C 0.000} C_DIS
LIN {X -63.134,Y 14.287,Z -11.294,A 90.000,B 90.000,C 0.000} C_DIS
LIN {X -65.956,Y 14.287,Z -10.104,A 90.000,B 90.000,C 0.000} C_DIS
LIN {X -68.756,Y 14.287,Z -8.864,A 90.000,B 90.000,C 0.000} C_DIS
LIN {X -69.854,Y 14.287,Z -8.335,A 90.000,B 90.000,C 0.000} C_DIS
LIN {X -70.978,Y 14.287,Z -7.865,A 90.000,B 90.000,C 0.000} C_DIS
LIN {X -72.126,Y 14.287,Z -7.457,A 90.000,B 90.000,C 0.000} C_DIS
LIN {X -73.295,Y 14.287,Z -7.110,A 90.000,B 90.000,C 0.000} C_DIS
LIN {X -74.480,Y 14.287,Z -6.826,A 90.000,B 90.000,C 0.000} C_DIS
LIN {X -75.679,Y 14.287,Z -6.606,A 90.000,B 90.000,C 0.000} C_DIS
LIN {X -76.887,Y 14.287,Z -6.450,A 90.000,B 90.000,C 0.000} C_DIS
LIN {X -78.103,Y 14.287,Z -6.359,A 90.000,B 90.000,C 0.000} C_DIS
LIN {X -79.321,Y 14.287,Z -6.334,A 90.000,B 90.000,C 0.000} C_DIS
LIN {X -80.539,Y 14.287,Z -6.373,A 90.000,B 90.000,C 0.000} C_DIS
LIN {X -81.753,Y 14.287,Z -6.478,A 90.000,B 90.000,C 0.000} C_DIS
LIN {X -82.960,Y 14.287,Z -6.647,A 90.000,B 90.000,C 0.000} C_DIS
LIN {X -84.156,Y 14.287,Z -6.881,A 90.000,B 90.000,C 0.000} C_DIS
LIN {X -84.961,Y 14.287,Z -7.040,A 90.000,B 90.000,C 0.000} C_DIS
LIN {X -85.755,Y 14.287,Z -7.248,A 90.000,B 90.000,C 0.000} C_DIS
LIN {X -86.535,Y 14.287,Z -7.504,A 90.000,B 90.000,C 0.000} C_DIS
LIN {X -87.298,Y 14.287,Z -7.806,A 90.000,B 90.000,C 0.000} C_DIS
LIN {X -88.041,Y 14.287,Z -8.154,A 90.000,B 90.000,C 0.000} C_DIS
LIN {X -88.761,Y 14.287,Z -8.547,A 90.000,B 90.000,C 0.000} C_DIS
LIN {X -89.457,Y 14.287,Z -8.982,A 90.000,B 90.000,C 0.000} C_DIS
LIN {X -90.658,Y 14.287,Z -9.041,A 90.000,B 90.000,C 0.000} C_DIS
LIN {X -91.853,Y 14.287,Z -9.168,A 90.000,B 90.000,C 0.000} C_DIS
LIN {X -93.040,Y 14.287,Z -9.361,A 90.000,B 90.000,C 0.000} C_DIS
LIN {X -94.214,Y 14.287,Z -9.619,A 90.000,B 90.000,C 0.000} C_DIS
LIN {X -95.371,Y 14.287,Z -9.943,A 90.000,B 90.000,C 0.000} C_DIS
LIN {X -96.509,Y 14.287,Z -10.331,A 90.000,B 90.000,C 0.000} C_DIS
LIN {X -96.645,Y 14.287,Z -10.387,A 90.000,B 90.000,C 0.000} C_DIS
LIN {X -97.481,Y 14.287,Z -10.765,A 90.000,B 90.000,C 0.000} C_DIS
LIN {X -98.293,Y 14.287,Z -11.190,A 90.000,B 90.000,C 0.000} C_DIS
LIN {X -99.080,Y 14.287,Z -11.662,A 90.000,B 90.000,C 0.000} C_DIS
LIN {X -99.839,Y 14.287,Z -12.177,A 90.000,B 90.000,C 0.000} C_DIS
LIN {X -100.563,Y 14.287,Z -12.778,A 90.000,B 90.000,C 0.000} C_DIS
LIN {X -101.300,Y 14.287,Z -13.364,A 90.000,B 90.000,C 0.000} C_DIS
LIN {X -102.049,Y 14.287,Z -13.933,A 90.000,B 90.000,C 0.000} C_DIS
LIN {X -102.843,Y 14.287,Z -14.328,A 90.000,B 90.000,C 0.000} C_DIS
LIN {X -103.604,Y 14.287,Z -14.782,A 90.000,B 90.000,C 0.000} C_DIS
LIN {X -104.328,Y 14.287,Z -15.295,A 90.000,B 90.000,C 0.000} C_DIS
LIN {X -105.010,Y 14.287,Z -15.861,A 90.000,B 90.000,C 0.000} C_DIS
LIN {X -105.647,Y 14.287,Z -16.478,A 90.000,B 90.000,C 0.000} C_DIS
LIN {X -106.234,Y 14.287,Z -17.143,A 90.000,B 90.000,C 0.000} C_DIS
LIN {X -106.767,Y 14.287,Z -17.851,A 90.000,B 90.000,C 0.000} C_DIS
LIN {X -107.879,Y 14.287,Z -18.181,A 90.000,B 90.000,C 0.000} C_DIS
LIN {X -108.971,Y 14.287,Z -18.573,A 90.000,B 90.000,C 0.000} C_DIS
LIN {X -110.039,Y 14.287,Z -19.027,A 90.000,B 90.000,C 0.000} C_DIS
LIN {X -111.079,Y 14.287,Z -19.540,A 90.000,B 90.000,C 0.000} C_DIS
LIN {X -112.089,Y 14.287,Z -20.111,A 90.000,B 90.000,C 0.000} C_DIS
LIN {X -113.065,Y 14.287,Z -20.739,A 90.000,B 90.000,C 0.000} C_DIS
LIN {X -114.004,Y 14.287,Z -21.420,A 90.000,B 90.000,C 0.000} C_DIS
LIN {X -114.902,Y 14.287,Z -22.154,A 90.000,B 90.000,C 0.000} C_DIS
LIN {X -115.758,Y 14.287,Z -22.937,A 90.000,B 90.000,C 0.000} C_DIS
LIN {X -116.568,Y 14.287,Z -23.768,A 90.000,B 90.000,C 0.000} C_DIS
LIN {X -117.330,Y 14.287,Z -24.643,A 90.000,B 90.000,C 0.000} C_DIS
LIN {X -117.877,Y 14.287,Z -25.450,A 90.000,B 90.000,C 0.000} C_DIS
LIN {X -118.467,Y 14.287,Z -26.225,A 90.000,B 90.000,C 0.000} C_DIS
LIN {X -119.099,Y 14.287,Z -26.967,A 90.000,B 90.000,C 0.000} C_DIS
LIN {X -119.770,Y 14.287,Z -27.674,A 90.000,B 90.000,C 0.000} C_DIS
LIN {X -120.392,Y 14.287,Z -28.586,A 90.000,B 90.000,C 0.000} C_DIS
LIN {X -120.953,Y 14.287,Z -29.537,A 90.000,B 90.000,C 0.000} C_DIS
LIN {X -121.449,Y 14.287,Z -30.524,A 90.000,B 90.000,C 0.000} C_DIS
LIN {X -121.878,Y 14.287,Z -31.541,A 90.000,B 90.000,C 0.000} C_DIS
LIN {X -122.239,Y 14.287,Z -32.584,A 90.000,B 90.000,C 0.000} C_DIS
LIN {X -122.529,Y 14.287,Z -33.649,A 90.000,B 90.000,C 0.000} C_DIS
LIN {X -122.749,Y 14.287,Z -34.732,A 90.000,B 90.000,C 0.000} C_DIS
LIN {X -122.895,Y 14.287,Z -35.826,A 90.000,B 90.000,C 0.000} C_DIS
LIN {X -122.969,Y 14.287,Z -36.927,A 90.000,B 90.000,C 0.000} C_DIS
LIN {X -122.970,Y 14.287,Z -38.031,A 90.000,B 90.000,C 0.000} C_DIS
LIN {X -122.897,Y 14.287,Z -39.133,A 90.000,B 90.000,C 0.000} C_DIS
LIN {X -122.751,Y 14.287,Z -40.228,A 90.000,B 90.000,C 0.000} C_DIS
LIN {X -122.532,Y 14.287,Z -41.310,A 90.000,B 90.000,C 0.000} C_DIS
LIN {X -122.243,Y 14.287,Z -42.375,A 90.000,B 90.000,C 0.000} C_DIS
LIN {X -121.883,Y 14.287,Z -43.419,A 90.000,B 90.000,C 0.000} C_DIS
LIN {X -122.053,Y 14.287,Z -44.374,A 90.000,B 90.000,C 0.000} C_DIS
LIN {X -122.161,Y 14.287,Z -45.338,A 90.000,B 90.000,C 0.000} C_DIS
LIN {X -122.207,Y 14.287,Z -46.307,A 90.000,B 90.000,C 0.000} C_DIS
LIN {X -122.191,Y 14.287,Z -47.277,A 90.000,B 90.000,C 0.000} C_DIS
LIN {X -122.111,Y 14.287,Z -48.244,A 90.000,B 90.000,C 0.000} C_DIS
LIN {X -121.970,Y 14.287,Z -49.204,A 90.000,B 90.000,C 0.000} C_DIS
LIN {X -121.767,Y 14.287,Z -50.153,A 90.000,B 90.000,C 0.000} C_DIS
LIN {X -121.504,Y 14.287,Z -51.086,A 90.000,B 90.000,C 0.000} C_DIS
LIN {X -121.181,Y 14.287,Z -52.001,A 90.000,B 90.000,C 0.000} C_DIS
LIN {X -120.799,Y 14.287,Z -52.893,A 90.000,B 90.000,C 0.000} C_DIS
LIN {X -120.485,Y 14.287,Z -54.139,A 90.000,B 90.000,C 0.000} C_DIS
LIN {X -120.143,Y 14.287,Z -55.377,A 90.000,B 90.000,C 0.000} C_DIS
LIN {X -119.772,Y 14.287,Z -56.607,A 90.000,B 90.000,C 0.000} C_DIS
LIN {X -119.454,Y 14.287,Z -58.085,A 90.000,B 90.000,C 0.000} C_DIS
LIN {X -119.069,Y 14.287,Z -59.546,A 90.000,B 90.000,C 0.000} C_DIS
LIN {X -118.617,Y 14.287,Z -60.988,A 90.000,B 90.000,C 0.000} C_DIS
LIN {X -118.100,Y 14.287,Z -62.408,A 90.000,B 90.000,C 0.000} C_DIS
LIN {X -117.518,Y 14.287,Z -63.803,A 90.000,B 90.000,C 0.000} C_DIS
LIN {X -116.873,Y 14.287,Z -65.170,A 90.000,B 90.000,C 0.000} C_DIS
LIN {X -116.165,Y 14.287,Z -66.506,A 90.000,B 90.000,C 0.000} C_DIS
LIN {X -115.398,Y 14.287,Z -67.808,A 90.000,B 90.000,C 0.000} C_DIS
LIN {X -114.571,Y 14.287,Z -69.073,A 90.000,B 90.000,C 0.000} C_DIS
LIN {X -113.687,Y 14.287,Z -70.299,A 90.000,B 90.000,C 0.000} C_DIS
LIN {X -112.748,Y 14.287,Z -71.483,A 90.000,B 90.000,C 0.000} C_DIS
LIN {X -111.756,Y 14.287,Z -72.623,A 90.000,B 90.000,C 0.000} C_DIS
LIN {X -110.712,Y 14.287,Z -73.717,A 90.000,B 90.000,C 0.000} C_DIS
LIN {X -109.620,Y 14.287,Z -74.761,A 90.000,B 90.000,C 0.000} C_DIS
LIN {X -108.894,Y 14.287,Z -75.489,A 90.000,B 90.000,C 0.000} C_DIS
LIN {X -108.128,Y 14.287,Z -76.175,A 90.000,B 90.000,C 0.000} C_DIS
LIN {X -107.324,Y 14.287,Z -76.815,A 90.000,B 90.000,C 0.000} C_DIS
LIN {X -106.484,Y 14.287,Z -77.407,A 90.000,B 90.000,C 0.000} C_DIS
LIN {X -105.611,Y 14.287,Z -77.951,A 90.000,B 90.000,C 0.000} C_DIS
LIN {X -104.709,Y 14.287,Z -78.444,A 90.000,B 90.000,C 0.000} C_DIS
LIN {X -103.780,Y 14.287,Z -78.884,A 90.000,B 90.000,C 0.000} C_DIS
LIN {X -103.652,Y 14.287,Z -78.952,A 90.000,B 90.000,C 0.000} C_DIS
LIN {X -102.856,Y 14.287,Z -79.358,A 90.000,B 90.000,C 0.000} C_DIS
LIN {X -102.037,Y 14.287,Z -79.716,A 90.000,B 90.000,C 0.000} C_DIS
LIN {X -101.198,Y 14.287,Z -80.024,A 90.000,B 90.000,C 0.000} C_DIS
LIN {X -100.343,Y 14.287,Z -80.283,A 90.000,B 90.000,C 0.000} C_DIS
LIN {X -99.473,Y 14.287,Z -80.490,A 90.000,B 90.000,C 0.000} C_DIS
LIN {X -98.593,Y 14.287,Z -80.645,A 90.000,B 90.000,C 0.000} C_DIS
LIN {X -98.439,Y 14.287,Z -80.681,A 90.000,B 90.000,C 0.000} C_DIS
LIN {X -96.737,Y 14.287,Z -80.917,A 90.000,B 90.000,C 0.000} C_DIS
LIN {X -95.031,Y 14.287,Z -81.118,A 90.000,B 90.000,C 0.000} C_DIS
LIN {X -93.321,Y 14.287,Z -81.286,A 90.000,B 90.000,C 0.000} C_DIS
LIN {X -93.146,Y 14.287,Z -81.314,A 90.000,B 90.000,C 0.000} C_DIS
LIN {X -92.593,Y 14.287,Z -81.517,A 90.000,B 90.000,C 0.000} C_DIS
LIN {X -92.058,Y 14.287,Z -81.764,A 90.000,B 90.000,C 0.000} C_DIS
LIN {X -91.545,Y 14.287,Z -82.055,A 90.000,B 90.000,C 0.000} C_DIS
LIN {X -91.059,Y 14.287,Z -82.388,A 90.000,B 90.000,C 0.000} C_DIS
LIN {X -89.751,Y 14.287,Z -83.565,A 90.000,B 90.000,C 0.000} C_DIS
LIN {X -88.408,Y 14.287,Z -84.701,A 90.000,B 90.000,C 0.000} C_DIS
LIN {X -87.030,Y 14.287,Z -85.794,A 90.000,B 90.000,C 0.000} C_DIS
LIN {X -85.619,Y 14.287,Z -86.845,A 90.000,B 90.000,C 0.000} C_DIS
LIN {X -84.177,Y 14.287,Z -87.853,A 90.000,B 90.000,C 0.000} C_DIS
LIN {X -82.704,Y 14.287,Z -88.815,A 90.000,B 90.000,C 0.000} C_DIS
LIN {X -80.158,Y 14.287,Z -90.417,A 90.000,B 90.000,C 0.000} C_DIS
LIN {X -77.625,Y 14.287,Z -92.039,A 90.000,B 90.000,C 0.000} C_DIS
LIN {X -76.194,Y 14.287,Z -92.933,A 90.000,B 90.000,C 0.000} C_DIS
LIN {X -74.799,Y 14.287,Z -93.880,A 90.000,B 90.000,C 0.000} C_DIS
LIN {X -73.441,Y 14.287,Z -94.880,A 90.000,B 90.000,C 0.000} C_DIS
LIN {X -72.121,Y 14.287,Z -95.931,A 90.000,B 90.000,C 0.000} C_DIS
LIN {X -70.843,Y 14.287,Z -97.032,A 90.000,B 90.000,C 0.000} C_DIS
LIN {X -69.608,Y 14.287,Z -98.180,A 90.000,B 90.000,C 0.000} C_DIS
LIN {X -68.417,Y 14.287,Z -99.375,A 90.000,B 90.000,C 0.000} C_DIS
LIN {X -67.273,Y 14.287,Z -100.614,A 90.000,B 90.000,C 0.000} C_DIS
LIN {X -66.177,Y 14.287,Z -101.897,A 90.000,B 90.000,C 0.000} C_DIS
LIN {X -65.130,Y 14.287,Z -103.219,A 90.000,B 90.000,C 0.000} C_DIS
LIN {X -63.219,Y 14.287,Z -105.846,A 90.000,B 90.000,C 0.000} C_DIS
LIN {X -61.276,Y 14.287,Z -108.449,A 90.000,B 90.000,C 0.000} C_DIS
LIN {X -59.300,Y 14.287,Z -111.027,A 90.000,B 90.000,C 0.000} C_DIS
LIN {X -57.292,Y 14.287,Z -113.581,A 90.000,B 90.000,C 0.000} C_DIS
LIN {X -55.252,Y 14.287,Z -116.109,A 90.000,B 90.000,C 0.000} C_DIS
LIN {X -53.905,Y 14.287,Z -117.618,A 90.000,B 90.000,C 0.000} C_DIS
LIN {X -52.602,Y 14.287,Z -119.166,A 90.000,B 90.000,C 0.000} C_DIS
LIN {X -51.345,Y 14.287,Z -120.751,A 90.000,B 90.000,C 0.000} C_DIS
LIN {X -50.134,Y 14.287,Z -122.372,A 90.000,B 90.000,C 0.000} C_DIS
LIN {X -48.971,Y 14.287,Z -124.028,A 90.000,B 90.000,C 0.000} C_DIS
LIN {X -48.160,Y 14.287,Z -125.670,A 90.000,B 90.000,C 0.000} C_DIS
LIN {X -47.389,Y 14.287,Z -127.330,A 90.000,B 90.000,C 0.000} C_DIS
LIN {X -46.658,Y 14.287,Z -129.010,A 90.000,B 90.000,C 0.000} C_DIS
LIN {X -45.969,Y 14.287,Z -130.706,A 90.000,B 90.000,C 0.000} C_DIS
LIN {X -45.181,Y 14.287,Z -132.612,A 90.000,B 90.000,C 0.000} C_DIS
LIN {X -44.337,Y 14.287,Z -134.494,A 90.000,B 90.000,C 0.000} C_DIS
LIN {X -43.438,Y 14.287,Z -136.350,A 90.000,B 90.000,C 0.000} C_DIS
LIN {X -42.485,Y 14.287,Z -138.179,A 90.000,B 90.000,C 0.000} C_DIS
LIN {X -41.477,Y 14.287,Z -139.979,A 90.000,B 90.000,C 0.000} C_DIS
LIN {X -40.417,Y 14.287,Z -141.748,A 90.000,B 90.000,C 0.000} C_DIS
LIN {X -39.305,Y 14.287,Z -143.485,A 90.000,B 90.000,C 0.000} C_DIS
LIN {X -38.142,Y 14.287,Z -145.188,A 90.000,B 90.000,C 0.000} C_DIS
LIN {X -36.929,Y 14.287,Z -146.856,A 90.000,B 90.000,C 0.000} C_DIS
LIN {X -35.667,Y 14.287,Z -148.488,A 90.000,B 90.000,C 0.000} C_DIS
LIN {X -34.357,Y 14.287,Z -150.081,A 90.000,B 90.000,C 0.000} C_DIS
LIN {X -32.177,Y 14.287,Z -152.435,A 90.000,B 90.000,C 0.000} C_DIS
LIN {X -29.965,Y 14.287,Z -154.761,A 90.000,B 90.000,C 0.000} C_DIS
LIN {X -27.722,Y 14.287,Z -157.056,A 90.000,B 90.000,C 0.000} C_DIS
LIN {X -25.449,Y 14.287,Z -159.321,A 90.000,B 90.000,C 0.000} C_DIS
LIN {X -24.833,Y 14.287,Z -159.908,A 90.000,B 90.000,C 0.000} C_DIS
LIN {X -24.254,Y 14.287,Z -160.532,A 90.000,B 90.000,C 0.000} C_DIS
LIN {X -23.714,Y 14.287,Z -161.190,A 90.000,B 90.000,C 0.000} C_DIS
LIN {X -23.215,Y 14.287,Z -161.879,A 90.000,B 90.000,C 0.000} C_DIS
LIN {X -22.758,Y 14.287,Z -162.597,A 90.000,B 90.000,C 0.000} C_DIS
LIN {X -23.115,Y 14.287,Z -163.460,A 90.000,B 90.000,C 0.000} C_DIS
LIN {X -23.519,Y 14.287,Z -164.302,A 90.000,B 90.000,C 0.000} C_DIS
LIN {X -23.968,Y 14.287,Z -165.121,A 90.000,B 90.000,C 0.000} C_DIS
LIN {X -24.780,Y 14.287,Z -166.407,A 90.000,B 90.000,C 0.000} C_DIS
LIN {X -25.640,Y 14.287,Z -167.662,A 90.000,B 90.000,C 0.000} C_DIS
LIN {X -26.544,Y 14.287,Z -168.885,A 90.000,B 90.000,C 0.000} C_DIS
LIN {X -27.494,Y 14.287,Z -170.073,A 90.000,B 90.000,C 0.000} C_DIS
LIN {X -28.486,Y 14.287,Z -171.226,A 90.000,B 90.000,C 0.000} C_DIS
LIN {X -29.520,Y 14.287,Z -172.342,A 90.000,B 90.000,C 0.000} C_DIS
LIN {X -30.594,Y 14.287,Z -173.419,A 90.000,B 90.000,C 0.000} C_DIS
LIN {X -31.707,Y 14.287,Z -174.455,A 90.000,B 90.000,C 0.000} C_DIS
LIN {X -32.858,Y 14.287,Z -175.450,A 90.000,B 90.000,C 0.000} C_DIS
LIN {X -35.875,Y 14.287,Z -177.819,A 90.000,B 90.000,C 0.000} C_DIS
LIN {X -38.929,Y 14.287,Z -180.140,A 90.000,B 90.000,C 0.000} C_DIS
LIN {X -42.019,Y 14.287,Z -182.413,A 90.000,B 90.000,C 0.000} C_DIS
LIN {X -45.144,Y 14.287,Z -184.637,A 90.000,B 90.000,C 0.000} C_DIS
LIN {X -48.303,Y 14.287,Z -186.813,A 90.000,B 90.000,C 0.000} C_DIS
LIN {X -51.496,Y 14.287,Z -188.938,A 90.000,B 90.000,C 0.000} C_DIS
LIN {X -54.722,Y 14.287,Z -191.013,A 90.000,B 90.000,C 0.000} C_DIS
LIN {X -57.980,Y 14.287,Z -193.038,A 90.000,B 90.000,C 0.000} C_DIS
LIN {X -61.453,Y 14.287,Z -195.127,A 90.000,B 90.000,C 0.000} C_DIS
LIN {X -64.912,Y 14.287,Z -197.237,A 90.000,B 90.000,C 0.000} C_DIS
LIN {X -70.964,Y 14.287,Z -200.799,A 90.000,B 90.000,C 0.000} C_DIS
LIN {X -76.988,Y 14.287,Z -204.408,A 90.000,B 90.000,C 0.000} C_DIS
LIN {X -82.985,Y 14.287,Z -208.062,A 90.000,B 90.000,C 0.000} C_DIS
LIN {X -88.954,Y 14.287,Z -211.761,A 90.000,B 90.000,C 0.000} C_DIS
LIN {X -94.895,Y 14.287,Z -215.506,A 90.000,B 90.000,C 0.000} C_DIS
LIN {X -100.807,Y 14.287,Z -219.296,A 90.000,B 90.000,C 0.000} C_DIS
LIN {X -106.690,Y 14.287,Z -223.130,A 90.000,B 90.000,C 0.000} C_DIS
LIN {X -114.380,Y 14.287,Z -228.216,A 90.000,B 90.000,C 0.000} C_DIS
LIN {X -121.778,Y 14.287,Z -233.180,A 90.000,B 90.000,C 0.000} C_DIS
LIN {X -128.845,Y 14.287,Z -237.978,A 90.000,B 90.000,C 0.000} C_DIS
LIN {X -135.503,Y 14.287,Z -242.529,A 90.000,B 90.000,C 0.000} C_DIS
LIN {X -136.644,Y 14.287,Z -243.489,A 90.000,B 90.000,C 0.000} C_DIS
LIN {X -136.709,Y 14.287,Z -243.561,A 90.000,B 90.000,C 0.000} C_DIS
LIN {X -145.015,Y 14.287,Z -243.561,A 90.000,B 90.000,C 0.000} C_DIS
LIN {X -145.015,Y 14.287,Z 0.000,A 90.000,B 90.000,C 0.000} C_DIS
LIN {X 145.015,Y 14.287,Z 0.000,A 90.000,B 90.000,C 0.000} C_DIS
LIN {X 145.015,Y 14.287,Z -243.561,A 90.000,B 90.000,C 0.000} C_DIS
LIN {X 98.929,Y 14.287,Z -243.561,A 90.000,B 90.000,C 0.000} C_DIS
LIN {X 100.061,Y 14.287,Z -240.011,A 90.000,B 90.000,C 0.000} C_DIS
LIN {X 101.151,Y 14.287,Z -236.449,A 90.000,B 90.000,C 0.000} C_DIS
LIN {X 102.200,Y 14.287,Z -232.874,A 90.000,B 90.000,C 0.000} C_DIS
LIN {X 103.208,Y 14.287,Z -229.287,A 90.000,B 90.000,C 0.000} C_DIS
LIN {X 104.581,Y 14.287,Z -223.630,A 90.000,B 90.000,C 0.000} C_DIS
LIN {X 105.883,Y 14.287,Z -217.956,A 90.000,B 90.000,C 0.000} C_DIS
LIN {X 107.115,Y 14.287,Z -212.267,A 90.000,B 90.000,C 0.000} C_DIS
LIN {X 108.276,Y 14.287,Z -206.563,A 90.000,B 90.000,C 0.000} C_DIS
LIN {X 109.366,Y 14.287,Z -200.845,A 90.000,B 90.000,C 0.000} C_DIS
LIN {X 110.385,Y 14.287,Z -195.113,A 90.000,B 90.000,C 0.000} C_DIS
LIN {X 111.332,Y 14.287,Z -189.370,A 90.000,B 90.000,C 0.000} C_DIS
LIN {X 112.208,Y 14.287,Z -183.615,A 90.000,B 90.000,C 0.000} C_DIS
LIN {X 113.012,Y 14.287,Z -177.850,A 90.000,B 90.000,C 0.000} C_DIS
LIN {X 113.745,Y 14.287,Z -172.075,A 90.000,B 90.000,C 0.000} C_DIS
LIN {X 114.405,Y 14.287,Z -166.291,A 90.000,B 90.000,C 0.000} C_DIS
LIN {X 114.881,Y 14.287,Z -162.571,A 90.000,B 90.000,C 0.000} C_DIS
LIN {X 115.291,Y 14.287,Z -158.844,A 90.000,B 90.000,C 0.000} C_DIS
LIN {X 115.635,Y 14.287,Z -155.109,A 90.000,B 90.000,C 0.000} C_DIS
LIN {X 115.911,Y 14.287,Z -151.369,A 90.000,B 90.000,C 0.000} C_DIS
LIN {X 116.121,Y 14.287,Z -147.625,A 90.000,B 90.000,C 0.000} C_DIS
LIN {X 116.263,Y 14.287,Z -143.877,A 90.000,B 90.000,C 0.000} C_DIS
LIN {X 116.339,Y 14.287,Z -140.128,A 90.000,B 90.000,C 0.000} C_DIS
LIN {X 116.348,Y 14.287,Z -136.378,A 90.000,B 90.000,C 0.000} C_DIS
LIN {X 116.289,Y 14.287,Z -132.628,A 90.000,B 90.000,C 0.000} C_DIS
LIN {X 116.164,Y 14.287,Z -128.880,A 90.000,B 90.000,C 0.000} C_DIS
LIN {X 115.907,Y 14.287,Z -125.252,A 90.000,B 90.000,C 0.000} C_DIS
LIN {X 115.594,Y 14.287,Z -121.628,A 90.000,B 90.000,C 0.000} C_DIS
LIN {X 115.225,Y 14.287,Z -118.009,A 90.000,B 90.000,C 0.000} C_DIS
LIN {X 114.799,Y 14.287,Z -114.397,A 90.000,B 90.000,C 0.000} C_DIS
LIN {X 114.318,Y 14.287,Z -110.791,A 90.000,B 90.000,C 0.000} C_DIS
LIN {X 113.781,Y 14.287,Z -107.194,A 90.000,B 90.000,C 0.000} C_DIS
LIN {X 113.188,Y 14.287,Z -103.605,A 90.000,B 90.000,C 0.000} C_DIS
LIN {X 112.539,Y 14.287,Z -100.026,A 90.000,B 90.000,C 0.000} C_DIS
LIN {X 111.835,Y 14.287,Z -96.457,A 90.000,B 90.000,C 0.000} C_DIS
LIN {X 111.589,Y 14.287,Z -95.017,A 90.000,B 90.000,C 0.000} C_DIS
LIN {X 111.277,Y 14.287,Z -93.591,A 90.000,B 90.000,C 0.000} C_DIS
LIN {X 110.899,Y 14.287,Z -92.180,A 90.000,B 90.000,C 0.000} C_DIS
LIN {X 110.455,Y 14.287,Z -90.788,A 90.000,B 90.000,C 0.000} C_DIS
LIN {X 109.948,Y 14.287,Z -89.419,A 90.000,B 90.000,C 0.000} C_DIS
LIN {X 109.378,Y 14.287,Z -88.074,A 90.000,B 90.000,C 0.000} C_DIS
LIN {X 108.745,Y 14.287,Z -86.758,A 90.000,B 90.000,C 0.000} C_DIS
LIN {X 108.053,Y 14.287,Z -85.472,A 90.000,B 90.000,C 0.000} C_DIS
LIN {X 109.254,Y 14.287,Z -83.491,A 90.000,B 90.000,C 0.000} C_DIS
LIN {X 110.393,Y 14.287,Z -81.474,A 90.000,B 90.000,C 0.000} C_DIS
LIN {X 111.472,Y 14.287,Z -79.424,A 90.000,B 90.000,C 0.000} C_DIS
LIN {X 112.487,Y 14.287,Z -77.342,A 90.000,B 90.000,C 0.000} C_DIS
LIN {X 113.439,Y 14.287,Z -75.230,A 90.000,B 90.000,C 0.000} C_DIS
LIN {X 114.327,Y 14.287,Z -73.090,A 90.000,B 90.000,C 0.000} C_DIS
LIN {X 115.149,Y 14.287,Z -70.924,A 90.000,B 90.000,C 0.000} C_DIS
LIN {X 115.905,Y 14.287,Z -68.735,A 90.000,B 90.000,C 0.000} C_DIS
LIN {X 116.594,Y 14.287,Z -66.523,A 90.000,B 90.000,C 0.000} C_DIS
LIN {X 117.391,Y 14.287,Z -63.629,A 90.000,B 90.000,C 0.000} C_DIS
LIN {X 118.216,Y 14.287,Z -60.743,A 90.000,B 90.000,C 0.000} C_DIS
LIN {X 118.900,Y 14.287,Z -58.947,A 90.000,B 90.000,C 0.000} C_DIS
LIN {X 119.632,Y 14.287,Z -57.170,A 90.000,B 90.000,C 0.000} C_DIS
LIN {X 120.411,Y 14.287,Z -55.413,A 90.000,B 90.000,C 0.000} C_DIS
LIN {X 121.238,Y 14.287,Z -53.679,A 90.000,B 90.000,C 0.000} C_DIS
LIN {X 122.112,Y 14.287,Z -51.967,A 90.000,B 90.000,C 0.000} C_DIS
LIN {X 122.620,Y 14.287,Z -50.961,A 90.000,B 90.000,C 0.000} C_DIS
LIN {X 123.069,Y 14.287,Z -49.926,A 90.000,B 90.000,C 0.000} C_DIS
LIN {X 123.455,Y 14.287,Z -48.867,A 90.000,B 90.000,C 0.000} C_DIS
LIN {X 123.778,Y 14.287,Z -47.788,A 90.000,B 90.000,C 0.000} C_DIS
LIN {X 124.038,Y 14.287,Z -46.690,A 90.000,B 90.000,C 0.000} C_DIS
LIN {X 124.232,Y 14.287,Z -45.580,A 90.000,B 90.000,C 0.000} C_DIS
LIN {X 124.360,Y 14.287,Z -44.460,A 90.000,B 90.000,C 0.000} C_DIS
LIN {X 124.422,Y 14.287,Z -43.334,A 90.000,B 90.000,C 0.000} C_DIS
LIN {X 124.417,Y 14.287,Z -42.207,A 90.000,B 90.000,C 0.000} C_DIS
LIN {X 124.347,Y 14.287,Z -41.082,A 90.000,B 90.000,C 0.000} C_DIS
LIN {X 124.254,Y 14.287,Z -40.095,A 90.000,B 90.000,C 0.000} C_DIS
LIN {X 124.088,Y 14.287,Z -39.117,A 90.000,B 90.000,C 0.000} C_DIS
LIN {X 123.849,Y 14.287,Z -38.155,A 90.000,B 90.000,C 0.000} C_DIS
LIN {X 123.540,Y 14.287,Z -37.213,A 90.000,B 90.000,C 0.000} C_DIS
LIN {X 123.161,Y 14.287,Z -36.296,A 90.000,B 90.000,C 0.000} C_DIS
LIN {X 122.715,Y 14.287,Z -35.411,A 90.000,B 90.000,C 0.000} C_DIS
LIN {X 122.205,Y 14.287,Z -34.561,A 90.000,B 90.000,C 0.000} C_DIS
LIN {X 121.633,Y 14.287,Z -33.751,A 90.000,B 90.000,C 0.000} C_DIS
LIN {X 121.002,Y 14.287,Z -32.986,A 90.000,B 90.000,C 0.000} C_DIS
LIN {X 120.316,Y 14.287,Z -32.270,A 90.000,B 90.000,C 0.000} C_DIS
LIN {X 119.578,Y 14.287,Z -31.607,A 90.000,B 90.000,C 0.000} C_DIS
LIN {X 118.794,Y 14.287,Z -31.001,A 90.000,B 90.000,C 0.000} C_DIS
LIN {X 117.966,Y 14.287,Z -30.455,A 90.000,B 90.000,C 0.000} C_DIS
LIN {X 117.834,Y 14.287,Z -30.373,A 90.000,B 90.000,C 0.000} C_DIS
LIN {X 117.055,Y 14.287,Z -29.942,A 90.000,B 90.000,C 0.000} C_DIS
LIN {X 116.250,Y 14.287,Z -29.561,A 90.000,B 90.000,C 0.000} C_DIS
LIN {X 115.424,Y 14.287,Z -29.230,A 90.000,B 90.000,C 0.000} C_DIS
LIN {X 114.578,Y 14.287,Z -28.952,A 90.000,B 90.000,C 0.000} C_DIS
LIN {X 114.396,Y 14.287,Z -28.894,A 90.000,B 90.000,C 0.000} C_DIS
LIN {X 113.507,Y 14.287,Z -28.671,A 90.000,B 90.000,C 0.000} C_DIS
LIN {X 112.605,Y 14.287,Z -28.507,A 90.000,B 90.000,C 0.000} C_DIS
LIN {X 111.695,Y 14.287,Z -28.401,A 90.000,B 90.000,C 0.000} C_DIS
LIN {X 110.779,Y 14.287,Z -28.354,A 90.000,B 90.000,C 0.000} C_DIS
LIN {X 109.863,Y 14.287,Z -28.367,A 90.000,B 90.000,C 0.000} C_DIS
LIN {X 108.949,Y 14.287,Z -28.439,A 90.000,B 90.000,C 0.000} C_DIS
LIN {X 108.042,Y 14.287,Z -28.571,A 90.000,B 90.000,C 0.000} C_DIS
LIN {X 107.145,Y 14.287,Z -28.761,A 90.000,B 90.000,C 0.000} C_DIS
LIN {X 105.009,Y 14.287,Z -29.519,A 90.000,B 90.000,C 0.000} C_DIS
LIN {X 102.893,Y 14.287,Z -30.330,A 90.000,B 90.000,C 0.000} C_DIS
LIN {X 100.797,Y 14.287,Z -31.192,A 90.000,B 90.000,C 0.000} C_DIS
LIN {X 98.723,Y 14.287,Z -32.105,A 90.000,B 90.000,C 0.000} C_DIS
LIN {X 96.671,Y 14.287,Z -33.068,A 90.000,B 90.000,C 0.000} C_DIS
LIN {X 95.024,Y 14.287,Z -33.842,A 90.000,B 90.000,C 0.000} C_DIS
LIN {X 93.410,Y 14.287,Z -34.680,A 90.000,B 90.000,C 0.000} C_DIS
LIN {X 91.829,Y 14.287,Z -35.581,A 90.000,B 90.000,C 0.000} C_DIS
LIN {X 90.286,Y 14.287,Z -36.544,A 90.000,B 90.000,C 0.000} C_DIS
LIN {X 88.781,Y 14.287,Z -37.567,A 90.000,B 90.000,C 0.000} C_DIS
LIN {X 87.318,Y 14.287,Z -38.649,A 90.000,B 90.000,C 0.000} C_DIS
LIN {X 85.899,Y 14.287,Z -39.787,A 90.000,B 90.000,C 0.000} C_DIS
LIN {X 84.526,Y 14.287,Z -40.981,A 90.000,B 90.000,C 0.000} C_DIS
LIN {X 83.201,Y 14.287,Z -42.228,A 90.000,B 90.000,C 0.000} C_DIS
LIN {X 81.926,Y 14.287,Z -43.526,A 90.000,B 90.000,C 0.000} C_DIS
LIN {X 81.037,Y 14.287,Z -44.437,A 90.000,B 90.000,C 0.000} C_DIS
LIN {X 80.197,Y 14.287,Z -45.393,A 90.000,B 90.000,C 0.000} C_DIS
LIN {X 79.409,Y 14.287,Z -46.392,A 90.000,B 90.000,C 0.000} C_DIS
LIN {X 78.675,Y 14.287,Z -47.431,A 90.000,B 90.000,C 0.000} C_DIS
LIN {X 77.997,Y 14.287,Z -48.508,A 90.000,B 90.000,C 0.000} C_DIS
LIN {X 77.376,Y 14.287,Z -49.619,A 90.000,B 90.000,C 0.000} C_DIS
LIN {X 77.376,Y 26.788,Z -49.619,A 90.000,B 90.000,C 0.000} C_DIS
LIN {X 77.376,Y 39.288,Z -49.619,A 90.000,B 90.000,C 0.000} C_DIS
LIN {X 77.376,Y 58.395,Z -49.619,A 90.000,B 90.000,C 0.000} C_DIS
LIN {X 144.015,Y 58.395,Z -242.561,A 90.000,B 90.000,C 0.000} C_DIS
LIN {X 144.015,Y 32.144,Z -242.561,A 90.000,B 90.000,C 0.000} C_DIS
LIN {X 144.015,Y 19.644,Z -242.561,A 90.000,B 90.000,C 0.000} C_DIS
LIN {X 144.015,Y 7.144,Z -242.561,A 90.000,B 90.000,C 0.000} C_DIS
LIN {X 105.716,Y 7.144,Z -242.561,A 90.000,B 90.000,C 0.000} C_DIS
LIN {X 106.605,Y 7.144,Z -240.057,A 90.000,B 90.000,C 0.000} C_DIS
LIN {X 107.459,Y 7.144,Z -237.540,A 90.000,B 90.000,C 0.000} C_DIS
LIN {X 108.278,Y 7.144,Z -235.012,A 90.000,B 90.000,C 0.000} C_DIS
LIN {X 144.015,Y 7.144,Z -235.012,A 90.000,B 90.000,C 0.000} C_DIS
LIN {X 144.015,Y 7.144,Z -227.464,A 90.000,B 90.000,C 0.000} C_DIS
LIN {X 110.491,Y 7.144,Z -227.464,A 90.000,B 90.000,C 0.000} C_DIS
LIN {X 110.666,Y 7.144,Z -226.814,A 90.000,B 90.000,C 0.000} C_DIS
LIN {X 111.487,Y 7.144,Z -223.369,A 90.000,B 90.000,C 0.000} C_DIS
LIN {X 112.269,Y 7.144,Z -219.915,A 90.000,B 90.000,C 0.000} C_DIS
LIN {X 144.015,Y 7.144,Z -219.915,A 90.000,B 90.000,C 0.000} C_DIS
LIN {X 144.015,Y 7.144,Z -212.366,A 90.000,B 90.000,C 0.000} C_DIS
LIN {X 113.841,Y 7.144,Z -212.366,A 90.000,B 90.000,C 0.000} C_DIS
LIN {X 114.322,Y 7.144,Z -209.853,A 90.000,B 90.000,C 0.000} C_DIS
LIN {X 114.783,Y 7.144,Z -207.337,A 90.000,B 90.000,C 0.000} C_DIS
LIN {X 115.224,Y 7.144,Z -204.817,A 90.000,B 90.000,C 0.000} C_DIS
LIN {X 144.015,Y 7.144,Z -204.817,A 90.000,B 90.000,C 0.000} C_DIS
LIN {X 144.015,Y 7.144,Z -197.269,A 90.000,B 90.000,C 0.000} C_DIS
LIN {X 116.422,Y 7.144,Z -197.269,A 90.000,B 90.000,C 0.000} C_DIS
LIN {X 116.669,Y 7.144,Z -195.548,A 90.000,B 90.000,C 0.000} C_DIS
LIN {X 116.907,Y 7.144,Z -193.826,A 90.000,B 90.000,C 0.000} C_DIS
LIN {X 117.160,Y 7.144,Z -191.773,A 90.000,B 90.000,C 0.000} C_DIS
LIN {X 117.406,Y 7.144,Z -189.720,A 90.000,B 90.000,C 0.000} C_DIS
LIN {X 144.015,Y 7.144,Z -189.720,A 90.000,B 90.000,C 0.000} C_DIS
LIN {X 144.015,Y 7.144,Z -182.171,A 90.000,B 90.000,C 0.000} C_DIS
LIN {X 118.234,Y 7.144,Z -182.171,A 90.000,B 90.000,C 0.000} C_DIS
LIN {X 118.606,Y 7.144,Z -178.398,A 90.000,B 90.000,C 0.000} C_DIS
LIN {X 118.950,Y 7.144,Z -174.622,A 90.000,B 90.000,C 0.000} C_DIS
LIN {X 144.015,Y 7.144,Z -174.622,A 90.000,B 90.000,C 0.000} C_DIS
LIN {X 144.015,Y 7.144,Z -167.073,A 90.000,B 90.000,C 0.000} C_DIS
LIN {X 119.553,Y 7.144,Z -167.073,A 90.000,B 90.000,C 0.000} C_DIS
LIN {X 119.812,Y 7.144,Z -163.300,A 90.000,B 90.000,C 0.000} C_DIS
LIN {X 120.044,Y 7.144,Z -159.525,A 90.000,B 90.000,C 0.000} C_DIS
LIN {X 144.015,Y 7.144,Z -159.525,A 90.000,B 90.000,C 0.000} C_DIS
LIN {X 144.015,Y 7.144,Z -151.976,A 90.000,B 90.000,C 0.000} C_DIS
LIN {X 120.471,Y 7.144,Z -151.976,A 90.000,B 90.000,C 0.000} C_DIS
LIN {X 120.564,Y 7.144,Z -149.461,A 90.000,B 90.000,C 0.000} C_DIS
LIN {X 120.623,Y 7.144,Z -146.944,A 90.000,B 90.000,C 0.000} C_DIS
LIN {X 120.647,Y 7.144,Z -144.427,A 90.000,B 90.000,C 0.000} C_DIS
LIN {X 144.015,Y 7.144,Z -144.427,A 90.000,B 90.000,C 0.000} C_DIS
LIN {X 144.015,Y 7.144,Z -136.878,A 90.000,B 90.000,C 0.000} C_DIS
LIN {X 120.513,Y 7.144,Z -136.878,A 90.000,B 90.000,C 0.000} C_DIS
LIN {X 120.399,Y 7.144,Z -134.360,A 90.000,B 90.000,C 0.000} C_DIS
LIN {X 120.250,Y 7.144,Z -131.843,A 90.000,B 90.000,C 0.000} C_DIS
LIN {X 120.067,Y 7.144,Z -129.329,A 90.000,B 90.000,C 0.000} C_DIS
LIN {X 144.015,Y 7.144,Z -129.329,A 90.000,B 90.000,C 0.000} C_DIS
LIN {X 144.015,Y 7.144,Z -121.781,A 90.000,B 90.000,C 0.000} C_DIS
LIN {X 119.229,Y 7.144,Z -121.781,A 90.000,B 90.000,C 0.000} C_DIS
LIN {X 118.891,Y 7.144,Z -119.261,A 90.000,B 90.000,C 0.000} C_DIS
LIN {X 118.527,Y 7.144,Z -116.744,A 90.000,B 90.000,C 0.000} C_DIS
LIN {X 118.135,Y 7.144,Z -114.232,A 90.000,B 90.000,C 0.000} C_DIS
LIN {X 144.015,Y 7.144,Z -114.232,A 90.000,B 90.000,C 0.000} C_DIS
LIN {X 144.015,Y 7.144,Z -106.683,A 90.000,B 90.000,C 0.000} C_DIS
LIN {X 116.792,Y 7.144,Z -106.683,A 90.000,B 90.000,C 0.000} C_DIS
LIN {X 116.287,Y 7.144,Z -104.161,A 90.000,B 90.000,C 0.000} C_DIS
LIN {X 115.754,Y 7.144,Z -101.644,A 90.000,B 90.000,C 0.000} C_DIS
LIN {X 115.193,Y 7.144,Z -99.134,A 90.000,B 90.000,C 0.000} C_DIS
LIN {X 144.015,Y 7.144,Z -99.134,A 90.000,B 90.000,C 0.000} C_DIS
LIN {X 144.015,Y 7.144,Z -91.586,A 90.000,B 90.000,C 0.000} C_DIS
LIN {X 113.313,Y 7.144,Z -91.586,A 90.000,B 90.000,C 0.000} C_DIS
LIN {X 112.830,Y 7.144,Z -90.037,A 90.000,B 90.000,C 0.000} C_DIS
LIN {X 112.293,Y 7.144,Z -88.506,A 90.000,B 90.000,C 0.000} C_DIS
LIN {X 111.703,Y 7.144,Z -86.994,A 90.000,B 90.000,C 0.000} C_DIS
LIN {X 111.060,Y 7.144,Z -85.504,A 90.000,B 90.000,C 0.000} C_DIS
LIN {X 110.366,Y 7.144,Z -84.037,A 90.000,B 90.000,C 0.000} C_DIS
LIN {X 144.015,Y 7.144,Z -84.037,A 90.000,B 90.000,C 0.000} C_DIS
LIN {X 144.015,Y 7.144,Z -76.488,A 90.000,B 90.000,C 0.000} C_DIS
LIN {X 113.983,Y 7.144,Z -76.488,A 90.000,B 90.000,C 0.000} C_DIS
LIN {X 114.783,Y 7.144,Z -74.630,A 90.000,B 90.000,C 0.000} C_DIS
LIN {X 115.534,Y 7.144,Z -72.751,A 90.000,B 90.000,C 0.000} C_DIS
LIN {X 116.236,Y 7.144,Z -70.854,A 90.000,B 90.000,C 0.000} C_DIS
LIN {X 116.890,Y 7.144,Z -68.939,A 90.000,B 90.000,C 0.000} C_DIS
LIN {X 144.015,Y 7.144,Z -68.939,A 90.000,B 90.000,C 0.000} C_DIS
LIN {X 144.015,Y 7.144,Z -61.390,A 90.000,B 90.000,C 0.000} C_DIS
LIN {X 119.069,Y 7.144,Z -61.390,A 90.000,B 90.000,C 0.000} C_DIS
LIN {X 119.167,Y 7.144,Z -61.055,A 90.000,B 90.000,C 0.000} C_DIS
LIN {X 119.868,Y 7.144,Z -59.220,A 90.000,B 90.000,C 0.000} C_DIS
LIN {X 120.619,Y 7.144,Z -57.405,A 90.000,B 90.000,C 0.000} C_DIS
LIN {X 121.422,Y 7.144,Z -55.612,A 90.000,B 90.000,C 0.000} C_DIS
LIN {X 122.274,Y 7.144,Z -53.842,A 90.000,B 90.000,C 0.000} C_DIS
LIN {X 144.015,Y 7.144,Z -53.842,A 90.000,B 90.000,C 0.000} C_DIS
LIN {X 144.015,Y 7.144,Z -46.293,A 90.000,B 90.000,C 0.000} C_DIS
LIN {X 125.131,Y 7.144,Z -46.293,A 90.000,B 90.000,C 0.000} C_DIS
LIN {X 125.285,Y 7.144,Z -45.243,A 90.000,B 90.000,C 0.000} C_DIS
LIN {X 125.384,Y 7.144,Z -44.187,A 90.000,B 90.000,C 0.000} C_DIS
LIN {X 125.427,Y 7.144,Z -43.127,A 90.000,B 90.000,C 0.000} C_DIS
LIN {X 125.413,Y 7.144,Z -42.067,A 90.000,B 90.000,C 0.000} C_DIS
LIN {X 125.344,Y 7.144,Z -41.008,A 90.000,B 90.000,C 0.000} C_DIS
LIN {X 125.280,Y 7.144,Z -40.248,A 90.000,B 90.000,C 0.000} C_DIS
LIN {X 125.175,Y 7.144,Z -39.493,A 90.000,B 90.000,C 0.000} C_DIS
LIN {X 125.030,Y 7.144,Z -38.744,A 90.000,B 90.000,C 0.000} C_DIS
LIN {X 144.015,Y 7.144,Z -38.744,A 90.000,B 90.000,C 0.000} C_DIS
LIN {X 144.015,Y 7.144,Z -31.195,A 90.000,B 90.000,C 0.000} C_DIS
LIN {X 120.629,Y 7.144,Z -31.195,A 90.000,B 90.000,C 0.000} C_DIS
LIN {X 144.015,Y 7.144,Z -23.646,A 90.000,B 90.000,C 0.000} C_DIS
LIN {X 17.121,Y 7.144,Z -23.646,A 90.000,B 90.000,C 0.000} C_DIS
LIN {X 14.096,Y 7.144,Z -22.927,A 90.000,B 90.000,C 0.000} C_DIS
LIN {X 11.079,Y 7.144,Z -22.179,A 90.000,B 90.000,C 0.000} C_DIS
LIN {X 7.732,Y 7.144,Z -21.464,A 90.000,B 90.000,C 0.000} C_DIS
LIN {X 4.397,Y 7.144,Z -20.691,A 90.000,B 90.000,C 0.000} C_DIS
LIN {X 1.077,Y 7.144,Z -19.860,A 90.000,B 90.000,C 0.000} C_DIS
LIN {X -2.229,Y 7.144,Z -18.972,A 90.000,B 90.000,C 0.000} C_DIS
LIN {X -5.599,Y 7.144,Z -17.975,A 90.000,B 90.000,C 0.000} C_DIS
LIN {X -8.980,Y 7.144,Z -17.016,A 90.000,B 90.000,C 0.000} C_DIS
LIN {X -12.372,Y 7.144,Z -16.098,A 90.000,B 90.000,C 0.000} C_DIS
LIN {X 144.015,Y 7.144,Z -16.098,A 90.000,B 90.000,C 0.000} C_DIS
LIN {X 144.015,Y 7.144,Z -8.549,A 90.000,B 90.000,C 0.000} C_DIS
LIN {X -47.972,Y 7.144,Z -8.549,A 90.000,B 90.000,C 0.000} C_DIS
LIN {X -48.999,Y 7.144,Z -8.278,A 90.000,B 90.000,C 0.000} C_DIS
LIN {X -54.019,Y 7.144,Z -6.888,A 90.000,B 90.000,C 0.000} C_DIS
LIN {X -59.046,Y 7.144,Z -5.524,A 90.000,B 90.000,C 0.000} C_DIS
LIN {X -60.889,Y 7.144,Z -5.162,A 90.000,B 90.000,C 0.000} C_DIS
LIN {X -62.742,Y 7.144,Z -4.860,A 90.000,B 90.000,C 0.000} C_DIS
LIN {X -64.605,Y 7.144,Z -4.618,A 90.000,B 90.000,C 0.000} C_DIS
LIN {X -66.474,Y 7.144,Z -4.438,A 90.000,B 90.000,C 0.000} C_DIS
LIN {X -68.348,Y 7.144,Z -4.319,A 90.000,B 90.000,C 0.000} C_DIS
LIN {X -70.225,Y 7.144,Z -4.261,A 90.000,B 90.000,C 0.000} C_DIS
LIN {X -72.108,Y 7.144,Z -4.059,A 90.000,B 90.000,C 0.000} C_DIS
LIN {X -73.996,Y 7.144,Z -3.915,A 90.000,B 90.000,C 0.000} C_DIS
LIN {X -75.888,Y 7.144,Z -3.831,A 90.000,B 90.000,C 0.000} C_DIS
LIN {X -77.781,Y 7.144,Z -3.806,A 90.000,B 90.000,C 0.000} C_DIS
LIN {X -79.675,Y 7.144,Z -3.841,A 90.000,B 90.000,C 0.000} C_DIS
LIN {X -81.566,Y 7.144,Z -3.935,A 90.000,B 90.000,C 0.000} C_DIS
LIN {X -83.453,Y 7.144,Z -4.087,A 90.000,B 90.000,C 0.000} C_DIS
LIN {X -85.335,Y 7.144,Z -4.299,A 90.000,B 90.000,C 0.000} C_DIS
LIN {X -87.209,Y 7.144,Z -4.570,A 90.000,B 90.000,C 0.000} C_DIS
LIN {X -89.074,Y 7.144,Z -4.899,A 90.000,B 90.000,C 0.000} C_DIS
LIN {X -90.892,Y 7.144,Z -5.362,A 90.000,B 90.000,C 0.000} C_DIS
LIN {X -92.694,Y 7.144,Z -5.885,A 90.000,B 90.000,C 0.000} C_DIS
LIN {X -94.478,Y 7.144,Z -6.465,A 90.000,B 90.000,C 0.000} C_DIS
LIN {X -96.243,Y 7.144,Z -7.103,A 90.000,B 90.000,C 0.000} C_DIS
LIN {X -97.986,Y 7.144,Z -7.798,A 90.000,B 90.000,C 0.000} C_DIS
LIN {X -99.705,Y 7.144,Z -8.549,A 90.000,B 90.000,C 0.000} C_DIS
LIN {X -144.015,Y 7.144,Z -8.549,A 90.000,B 90.000,C 0.000} C_DIS
LIN {X -144.015,Y 7.144,Z -16.098,A 90.000,B 90.000,C 0.000} C_DIS
LIN {X -116.388,Y 7.144,Z -16.098,A 90.000,B 90.000,C 0.000} C_DIS
LIN {X -117.201,Y 7.144,Z -16.761,A 90.000,B 90.000,C 0.000} C_DIS
LIN {X -117.978,Y 7.144,Z -17.468,A 90.000,B 90.000,C 0.000} C_DIS
LIN {X -118.715,Y 7.144,Z -18.215,A 90.000,B 90.000,C 0.000} C_DIS
LIN {X -119.412,Y 7.144,Z -19.000,A 90.000,B 90.000,C 0.000} C_DIS
LIN {X -120.065,Y 7.144,Z -19.822,A 90.000,B 90.000,C 0.000} C_DIS
LIN {X -120.672,Y 7.144,Z -20.678,A 90.000,B 90.000,C 0.000} C_DIS
LIN {X -121.233,Y 7.144,Z -21.565,A 90.000,B 90.000,C 0.000} C_DIS
LIN {X -121.746,Y 7.144,Z -22.481,A 90.000,B 90.000,C 0.000} C_DIS
LIN {X -122.263,Y 7.144,Z -23.050,A 90.000,B 90.000,C 0.000} C_DIS
LIN {X -122.749,Y 7.144,Z -23.646,A 90.000,B 90.000,C 0.000} C_DIS
LIN {X -144.015,Y 7.144,Z -23.646,A 90.000,B 90.000,C 0.000} C_DIS
LIN {X -144.015,Y 7.144,Z -31.195,A 90.000,B 90.000,C 0.000} C_DIS
LIN {X -126.207,Y 7.144,Z -31.195,A 90.000,B 90.000,C 0.000} C_DIS
LIN {X -126.346,Y 7.144,Z -32.133,A 90.000,B 90.000,C 0.000} C_DIS
LIN {X -126.429,Y 7.144,Z -33.078,A 90.000,B 90.000,C 0.000} C_DIS
LIN {X -126.455,Y 7.144,Z -34.026,A 90.000,B 90.000,C 0.000} C_DIS
LIN {X -126.424,Y 7.144,Z -34.974,A 90.000,B 90.000,C 0.000} C_DIS
LIN {X -126.338,Y 7.144,Z -35.918,A 90.000,B 90.000,C 0.000} C_DIS
LIN {X -126.195,Y 7.144,Z -36.856,A 90.000,B 90.000,C 0.000} C_DIS
LIN {X -126.355,Y 7.144,Z -37.480,A 90.000,B 90.000,C 0.000} C_DIS
LIN {X -126.492,Y 7.144,Z -38.110,A 90.000,B 90.000,C 0.000} C_DIS
LIN {X -126.605,Y 7.144,Z -38.744,A 90.000,B 90.000,C 0.000} C_DIS
LIN {X -144.015,Y 7.144,Z -38.744,A 90.000,B 90.000,C 0.000} C_DIS
LIN {X -144.015,Y 7.144,Z -46.293,A 90.000,B 90.000,C 0.000} C_DIS
LIN {X -126.162,Y 7.144,Z -46.293,A 90.000,B 90.000,C 0.000} C_DIS
LIN {X -126.253,Y 7.144,Z -47.448,A 90.000,B 90.000,C 0.000} C_DIS
LIN {X -126.280,Y 7.144,Z -48.607,A 90.000,B 90.000,C 0.000} C_DIS
LIN {X -126.243,Y 7.144,Z -49.765,A 90.000,B 90.000,C 0.000} C_DIS
LIN {X -126.142,Y 7.144,Z -50.920,A 90.000,B 90.000,C 0.000} C_DIS
LIN {X -125.978,Y 7.144,Z -52.067,A 90.000,B 90.000,C 0.000} C_DIS
LIN {X -125.737,Y 7.144,Z -52.956,A 90.000,B 90.000,C 0.000} C_DIS
LIN {X -125.484,Y 7.144,Z -53.842,A 90.000,B 90.000,C 0.000} C_DIS
LIN {X -144.015,Y 7.144,Z -53.842,A 90.000,B 90.000,C 0.000} C_DIS
LIN {X -144.015,Y 7.144,Z -61.390,A 90.000,B 90.000,C 0.000} C_DIS
LIN {X -122.913,Y 7.144,Z -61.390,A 90.000,B 90.000,C 0.000} C_DIS
LIN {X -122.308,Y 7.144,Z -63.159,A 90.000,B 90.000,C 0.000} C_DIS
LIN {X -121.665,Y 7.144,Z -64.915,A 90.000,B 90.000,C 0.000} C_DIS
LIN {X -120.986,Y 7.144,Z -66.657,A 90.000,B 90.000,C 0.000} C_DIS
LIN {X -120.270,Y 7.144,Z -68.385,A 90.000,B 90.000,C 0.000} C_DIS
LIN {X -120.000,Y 7.144,Z -68.939,A 90.000,B 90.000,C 0.000} C_DIS
LIN {X -144.015,Y 7.144,Z -68.939,A 90.000,B 90.000,C 0.000} C_DIS
LIN {X -144.015,Y 7.144,Z -76.488,A 90.000,B 90.000,C 0.000} C_DIS
LIN {X -114.744,Y 7.144,Z -76.488,A 90.000,B 90.000,C 0.000} C_DIS
LIN {X -113.822,Y 7.144,Z -77.430,A 90.000,B 90.000,C 0.000} C_DIS
LIN {X -112.862,Y 7.144,Z -78.334,A 90.000,B 90.000,C 0.000} C_DIS
LIN {X -111.866,Y 7.144,Z -79.197,A 90.000,B 90.000,C 0.000} C_DIS
LIN {X -110.834,Y 7.144,Z -80.017,A 90.000,B 90.000,C 0.000} C_DIS
LIN {X -109.984,Y 7.144,Z -80.716,A 90.000,B 90.000,C 0.000} C_DIS
LIN {X -109.103,Y 7.144,Z -81.376,A 90.000,B 90.000,C 0.000} C_DIS
LIN {X -108.193,Y 7.144,Z -81.995,A 90.000,B 90.000,C 0.000} C_DIS
LIN {X -107.255,Y 7.144,Z -82.571,A 90.000,B 90.000,C 0.000} C_DIS
LIN {X -106.292,Y 7.144,Z -83.104,A 90.000,B 90.000,C 0.000} C_DIS
LIN {X -105.306,Y 7.144,Z -83.593,A 90.000,B 90.000,C 0.000} C_DIS
LIN {X -104.299,Y 7.144,Z -84.037,A 90.000,B 90.000,C 0.000} C_DIS
LIN {X -144.015,Y 7.144,Z -84.037,A 90.000,B 90.000,C 0.000} C_DIS
LIN {X -144.015,Y 7.144,Z -91.586,A 90.000,B 90.000,C 0.000} C_DIS
LIN {X -84.523,Y 7.144,Z -91.586,A 90.000,B 90.000,C 0.000} C_DIS
LIN {X -82.580,Y 7.144,Z -92.919,A 90.000,B 90.000,C 0.000} C_DIS
LIN {X -80.609,Y 7.144,Z -94.210,A 90.000,B 90.000,C 0.000} C_DIS
LIN {X -78.612,Y 7.144,Z -95.461,A 90.000,B 90.000,C 0.000} C_DIS
LIN {X -77.213,Y 7.144,Z -96.320,A 90.000,B 90.000,C 0.000} C_DIS
LIN {X -75.840,Y 7.144,Z -97.219,A 90.000,B 90.000,C 0.000} C_DIS
LIN {X -74.494,Y 7.144,Z -98.157,A 90.000,B 90.000,C 0.000} C_DIS
LIN {X -73.175,Y 7.144,Z -99.134,A 90.000,B 90.000,C 0.000} C_DIS
LIN {X -144.015,Y 7.144,Z -99.134,A 90.000,B 90.000,C 0.000} C_DIS
LIN {X -144.015,Y 7.144,Z -106.683,A 90.000,B 90.000,C 0.000} C_DIS
LIN {X -65.188,Y 7.144,Z -106.683,A 90.000,B 90.000,C 0.000} C_DIS
LIN {X -63.524,Y 7.144,Z -108.536,A 90.000,B 90.000,C 0.000} C_DIS
LIN {X -61.886,Y 7.144,Z -110.412,A 90.000,B 90.000,C 0.000} C_DIS
LIN {X -60.275,Y 7.144,Z -112.311,A 90.000,B 90.000,C 0.000} C_DIS
LIN {X -58.690,Y 7.144,Z -114.232,A 90.000,B 90.000,C 0.000} C_DIS
LIN {X -144.015,Y 7.144,Z -114.232,A 90.000,B 90.000,C 0.000} C_DIS
LIN {X -144.015,Y 7.144,Z -121.781,A 90.000,B 90.000,C 0.000} C_DIS
LIN {X -52.522,Y 7.144,Z -121.781,A 90.000,B 90.000,C 0.000} C_DIS
LIN {X -51.436,Y 7.144,Z -123.256,A 90.000,B 90.000,C 0.000} C_DIS
LIN {X -50.377,Y 7.144,Z -124.751,A 90.000,B 90.000,C 0.000} C_DIS
LIN {X -49.604,Y 7.144,Z -126.256,A 90.000,B 90.000,C 0.000} C_DIS
LIN {X -48.873,Y 7.144,Z -127.783,A 90.000,B 90.000,C 0.000} C_DIS
LIN {X -48.186,Y 7.144,Z -129.329,A 90.000,B 90.000,C 0.000} C_DIS
LIN {X -144.015,Y 7.144,Z -129.329,A 90.000,B 90.000,C 0.000} C_DIS
LIN {X -144.015,Y 7.144,Z -136.878,A 90.000,B 90.000,C 0.000} C_DIS
LIN {X -44.901,Y 7.144,Z -136.878,A 90.000,B 90.000,C 0.000} C_DIS
LIN {X -43.916,Y 7.144,Z -138.809,A 90.000,B 90.000,C 0.000} C_DIS
LIN {X -42.879,Y 7.144,Z -140.712,A 90.000,B 90.000,C 0.000} C_DIS
LIN {X -41.788,Y 7.144,Z -142.585,A 90.000,B 90.000,C 0.000} C_DIS
LIN {X -40.646,Y 7.144,Z -144.427,A 90.000,B 90.000,C 0.000} C_DIS
LIN {X -144.015,Y 7.144,Z -144.427,A 90.000,B 90.000,C 0.000} C_DIS
LIN {X -144.015,Y 7.144,Z -151.976,A 90.000,B 90.000,C 0.000} C_DIS
LIN {X -34.979,Y 7.144,Z -151.976,A 90.000,B 90.000,C 0.000} C_DIS
LIN {X -33.655,Y 7.144,Z -153.537,A 90.000,B 90.000,C 0.000} C_DIS
LIN {X -32.299,Y 7.144,Z -155.069,A 90.000,B 90.000,C 0.000} C_DIS
LIN {X -30.912,Y 7.144,Z -156.574,A 90.000,B 90.000,C 0.000} C_DIS
LIN {X -29.494,Y 7.144,Z -158.050,A 90.000,B 90.000,C 0.000} C_DIS
LIN {X -28.116,Y 7.144,Z -159.525,A 90.000,B 90.000,C 0.000} C_DIS
LIN {X -144.015,Y 7.144,Z -159.525,A 90.000,B 90.000,C 0.000} C_DIS
LIN {X -144.015,Y 7.144,Z -167.073,A 90.000,B 90.000,C 0.000} C_DIS
LIN {X -28.054,Y 7.144,Z -167.073,A 90.000,B 90.000,C 0.000} C_DIS
LIN {X -28.633,Y 7.144,Z -167.942,A 90.000,B 90.000,C 0.000} C_DIS
LIN {X -29.249,Y 7.144,Z -168.785,A 90.000,B 90.000,C 0.000} C_DIS
LIN {X -29.900,Y 7.144,Z -169.602,A 90.000,B 90.000,C 0.000} C_DIS
LIN {X -31.197,Y 7.144,Z -170.908,A 90.000,B 90.000,C 0.000} C_DIS
LIN {X -32.526,Y 7.144,Z -172.181,A 90.000,B 90.000,C 0.000} C_DIS
LIN {X -33.888,Y 7.144,Z -173.420,A 90.000,B 90.000,C 0.000} C_DIS
LIN {X -35.282,Y 7.144,Z -174.622,A 90.000,B 90.000,C 0.000} C_DIS
LIN {X -144.015,Y 7.144,Z -174.622,A 90.000,B 90.000,C 0.000} C_DIS
LIN {X -144.015,Y 7.144,Z -182.171,A 90.000,B 90.000,C 0.000} C_DIS
LIN {X -45.568,Y 7.144,Z -182.171,A 90.000,B 90.000,C 0.000} C_DIS
LIN {X -48.468,Y 7.144,Z -184.117,A 90.000,B 90.000,C 0.000} C_DIS
LIN {X -51.394,Y 7.144,Z -186.025,A 90.000,B 90.000,C 0.000} C_DIS
LIN {X -54.346,Y 7.144,Z -187.892,A 90.000,B 90.000,C 0.000} C_DIS
LIN {X -57.322,Y 7.144,Z -189.720,A 90.000,B 90.000,C 0.000} C_DIS
LIN {X -144.015,Y 7.144,Z -189.720,A 90.000,B 90.000,C 0.000} C_DIS
LIN {X -144.015,Y 7.144,Z -197.269,A 90.000,B 90.000,C 0.000} C_DIS
LIN {X -70.565,Y 7.144,Z -197.269,A 90.000,B 90.000,C 0.000} C_DIS
LIN {X -74.986,Y 7.144,Z -199.755,A 90.000,B 90.000,C 0.000} C_DIS
LIN {X -79.390,Y 7.144,Z -202.271,A 90.000,B 90.000,C 0.000} C_DIS
LIN {X -83.777,Y 7.144,Z -204.817,A 90.000,B 90.000,C 0.000} C_DIS
LIN {X -144.015,Y 7.144,Z -204.817,A 90.000,B 90.000,C 0.000} C_DIS
LIN {X -144.015,Y 7.144,Z -212.366,A 90.000,B 90.000,C 0.000} C_DIS
LIN {X -96.382,Y 7.144,Z -212.366,A 90.000,B 90.000,C 0.000} C_DIS
LIN {X -100.417,Y 7.144,Z -214.856,A 90.000,B 90.000,C 0.000} C_DIS
LIN {X -104.436,Y 7.144,Z -217.372,A 90.000,B 90.000,C 0.000} C_DIS
LIN {X -108.439,Y 7.144,Z -219.915,A 90.000,B 90.000,C 0.000} C_DIS
LIN {X -144.015,Y 7.144,Z -219.915,A 90.000,B 90.000,C 0.000} C_DIS
LIN {X -144.015,Y 7.144,Z -227.464,A 90.000,B 90.000,C 0.000} C_DIS
LIN {X -120.029,Y 7.144,Z -227.464,A 90.000,B 90.000,C 0.000} C_DIS
LIN {X -131.378,Y 7.144,Z -234.913,A 90.000,B 90.000,C 0.000} C_DIS
LIN {X -131.529,Y 7.144,Z -235.012,A 90.000,B 90.000,C 0.000} C_DIS
LIN {X -144.015,Y 7.144,Z -235.012,A 90.000,B 90.000,C 0.000} C_DIS
LIN {X -144.015,Y 7.144,Z -242.561,A 90.000,B 90.000,C 0.000} C_DIS
LIN {X -141.133,Y 7.144,Z -242.561,A 90.000,B 90.000,C 0.000} C_DIS
LIN {X -144.015,Y 7.144,Z -1.000,A 90.000,B 90.000,C 0.000} C_DIS
LIN {X 144.015,Y 7.144,Z -1.000,A 90.000,B 90.000,C 0.000} C_DIS
LIN {X 98.141,Y 7.144,Z -31.195,A 90.000,B 90.000,C 0.000} C_DIS
LIN {X 45.076,Y 7.144,Z -31.195,A 90.000,B 90.000,C 0.000} C_DIS
LIN {X 48.235,Y 7.144,Z -32.294,A 90.000,B 90.000,C 0.000} C_DIS
LIN {X 51.376,Y 7.144,Z -33.445,A 90.000,B 90.000,C 0.000} C_DIS
LIN {X 54.497,Y 7.144,Z -34.648,A 90.000,B 90.000,C 0.000} C_DIS
LIN {X 57.598,Y 7.144,Z -35.901,A 90.000,B 90.000,C 0.000} C_DIS
LIN {X 60.678,Y 7.144,Z -37.206,A 90.000,B 90.000,C 0.000} C_DIS
LIN {X 62.231,Y 7.144,Z -37.966,A 90.000,B 90.000,C 0.000} C_DIS
LIN {X 63.775,Y 7.144,Z -38.744,A 90.000,B 90.000,C 0.000} C_DIS
LIN {X 85.665,Y 7.144,Z -38.744,A 90.000,B 90.000,C 0.000} C_DIS
LIN {X 85.492,Y 7.144,Z -38.883,A 90.000,B 90.000,C 0.000} C_DIS
LIN {X 84.334,Y 7.144,Z -39.801,A 90.000,B 90.000,C 0.000} C_DIS
LIN {X 83.218,Y 7.144,Z -40.769,A 90.000,B 90.000,C 0.000} C_DIS
LIN {X 82.146,Y 7.144,Z -41.785,A 90.000,B 90.000,C 0.000} C_DIS
LIN {X 81.120,Y 7.144,Z -42.848,A 90.000,B 90.000,C 0.000} C_DIS
LIN {X 80.141,Y 7.144,Z -43.955,A 90.000,B 90.000,C 0.000} C_DIS
LIN {X 79.213,Y 7.144,Z -45.104,A 90.000,B 90.000,C 0.000} C_DIS
LIN {X 78.336,Y 7.144,Z -46.293,A 90.000,B 90.000,C 0.000} C_DIS
LIN {X 76.716,Y 7.144,Z -46.293,A 90.000,B 90.000,C 0.000} C_DIS
LIN {X 78.116,Y 7.144,Z -48.436,A 90.000,B 90.000,C 0.000} C_DIS
LIN {X 75.664,Y 7.144,Z -46.798,A 90.000,B 90.000,C 0.000} C_DIS
LIN {X 73.177,Y 7.144,Z -45.214,A 90.000,B 90.000,C 0.000} C_DIS
LIN {X 70.657,Y 7.144,Z -43.684,A 90.000,B 90.000,C 0.000} C_DIS
LIN {X 68.104,Y 7.144,Z -42.208,A 90.000,B 90.000,C 0.000} C_DIS
LIN {X 65.520,Y 7.144,Z -40.787,A 90.000,B 90.000,C 0.000} C_DIS
LIN {X 62.906,Y 7.144,Z -39.423,A 90.000,B 90.000,C 0.000} C_DIS
LIN {X 60.263,Y 7.144,Z -38.115,A 90.000,B 90.000,C 0.000} C_DIS
LIN {X 57.420,Y 7.144,Z -36.910,A 90.000,B 90.000,C 0.000} C_DIS
LIN {X 54.559,Y 7.144,Z -35.748,A 90.000,B 90.000,C 0.000} C_DIS
LIN {X 51.681,Y 7.144,Z -34.629,A 90.000,B 90.000,C 0.000} C_DIS
LIN {X 48.786,Y 7.144,Z -33.555,A 90.000,B 90.000,C 0.000} C_DIS
LIN {X 45.875,Y 7.144,Z -32.525,A 90.000,B 90.000,C 0.000} C_DIS
LIN {X 42.948,Y 7.144,Z -31.540,A 90.000,B 90.000,C 0.000} C_DIS
LIN {X 40.539,Y 7.144,Z -30.810,A 90.000,B 90.000,C 0.000} C_DIS
LIN {X 38.140,Y 7.144,Z -30.050,A 90.000,B 90.000,C 0.000} C_DIS
LIN {X 35.750,Y 7.144,Z -29.260,A 90.000,B 90.000,C 0.000} C_DIS
LIN {X 34.015,Y 7.144,Z -28.660,A 90.000,B 90.000,C 0.000} C_DIS
LIN {X 32.264,Y 7.144,Z -28.105,A 90.000,B 90.000,C 0.000} C_DIS
LIN {X 30.500,Y 7.144,Z -27.595,A 90.000,B 90.000,C 0.000} C_DIS
LIN {X 28.724,Y 7.144,Z -27.130,A 90.000,B 90.000,C 0.000} C_DIS
LIN {X 25.132,Y 7.144,Z -26.419,A 90.000,B 90.000,C 0.000} C_DIS
LIN {X 21.549,Y 7.144,Z -25.665,A 90.000,B 90.000,C 0.000} C_DIS
LIN {X 17.975,Y 7.144,Z -24.870,A 90.000,B 90.000,C 0.000} C_DIS
LIN {X 14.410,Y 7.144,Z -24.033,A 90.000,B 90.000,C 0.000} C_DIS
LIN {X 10.856,Y 7.144,Z -23.154,A 90.000,B 90.000,C 0.000} C_DIS
LIN {X 7.495,Y 7.144,Z -22.435,A 90.000,B 90.000,C 0.000} C_DIS
LIN {X 4.147,Y 7.144,Z -21.659,A 90.000,B 90.000,C 0.000} C_DIS
LIN {X 0.812,Y 7.144,Z -20.825,A 90.000,B 90.000,C 0.000} C_DIS
LIN {X -2.507,Y 7.144,Z -19.933,A 90.000,B 90.000,C 0.000} C_DIS
LIN {X -6.684,Y 7.144,Z -18.703,A 90.000,B 90.000,C 0.000} C_DIS
LIN {X -10.879,Y 7.144,Z -17.533,A 90.000,B 90.000,C 0.000} C_DIS
LIN {X -15.089,Y 7.144,Z -16.424,A 90.000,B 90.000,C 0.000} C_DIS
LIN {X -19.316,Y 7.144,Z -15.375,A 90.000,B 90.000,C 0.000} C_DIS
LIN {X -23.557,Y 7.144,Z -14.387,A 90.000,B 90.000,C 0.000} C_DIS
LIN {X -27.811,Y 7.144,Z -13.459,A 90.000,B 90.000,C 0.000} C_DIS
LIN {X -32.079,Y 7.144,Z -12.593,A 90.000,B 90.000,C 0.000} C_DIS
LIN {X -36.358,Y 7.144,Z -11.789,A 90.000,B 90.000,C 0.000} C_DIS
LIN {X -40.649,Y 7.144,Z -11.046,A 90.000,B 90.000,C 0.000} C_DIS
LIN {X -42.388,Y 7.144,Z -10.766,A 90.000,B 90.000,C 0.000} C_DIS
LIN {X -44.120,Y 7.144,Z -10.446,A 90.000,B 90.000,C 0.000} C_DIS
LIN {X -45.844,Y 7.144,Z -10.085,A 90.000,B 90.000,C 0.000} C_DIS
LIN {X -47.559,Y 7.144,Z -9.684,A 90.000,B 90.000,C 0.000} C_DIS
LIN {X -49.264,Y 7.144,Z -9.242,A 90.000,B 90.000,C 0.000} C_DIS
LIN {X -54.268,Y 7.144,Z -7.856,A 90.000,B 90.000,C 0.000} C_DIS
LIN {X -59.280,Y 7.144,Z -6.496,A 90.000,B 90.000,C 0.000} C_DIS
LIN {X -61.095,Y 7.144,Z -6.140,A 90.000,B 90.000,C 0.000} C_DIS
LIN {X -62.922,Y 7.144,Z -5.843,A 90.000,B 90.000,C 0.000} C_DIS
LIN {X -64.757,Y 7.144,Z -5.607,A 90.000,B 90.000,C 0.000} C_DIS
LIN {X -66.598,Y 7.144,Z -5.431,A 90.000,B 90.000,C 0.000} C_DIS
LIN {X -68.445,Y 7.144,Z -5.315,A 90.000,B 90.000,C 0.000} C_DIS
LIN {X -70.294,Y 7.144,Z -5.260,A 90.000,B 90.000,C 0.000} C_DIS
LIN {X -72.149,Y 7.144,Z -5.059,A 90.000,B 90.000,C 0.000} C_DIS
LIN {X -74.009,Y 7.144,Z -4.916,A 90.000,B 90.000,C 0.000} C_DIS
LIN {X -75.873,Y 7.144,Z -4.832,A 90.000,B 90.000,C 0.000} C_DIS
LIN {X -77.738,Y 7.144,Z -4.806,A 90.000,B 90.000,C 0.000} C_DIS
LIN {X -79.603,Y 7.144,Z -4.839,A 90.000,B 90.000,C 0.000} C_DIS
LIN {X -81.467,Y 7.144,Z -4.930,A 90.000,B 90.000,C 0.000} C_DIS
LIN {X -83.326,Y 7.144,Z -5.080,A 90.000,B 90.000,C 0.000} C_DIS
LIN {X -85.180,Y 7.144,Z -5.288,A 90.000,B 90.000,C 0.000} C_DIS
LIN {X -87.027,Y 7.144,Z -5.553,A 90.000,B 90.000,C 0.000} C_DIS
LIN {X -88.864,Y 7.144,Z -5.877,A 90.000,B 90.000,C 0.000} C_DIS
LIN {X -90.565,Y 7.144,Z -6.310,A 90.000,B 90.000,C 0.000} C_DIS
LIN {X -92.251,Y 7.144,Z -6.795,A 90.000,B 90.000,C 0.000} C_DIS
LIN {X -93.922,Y 7.144,Z -7.332,A 90.000,B 90.000,C 0.000} C_DIS
LIN {X -95.576,Y 7.144,Z -7.920,A 90.000,B 90.000,C 0.000} C_DIS
LIN {X -97.210,Y 7.144,Z -8.559,A 90.000,B 90.000,C 0.000} C_DIS
LIN {X -98.824,Y 7.144,Z -9.248,A 90.000,B 90.000,C 0.000} C_DIS
LIN {X -100.416,Y 7.144,Z -9.987,A 90.000,B 90.000,C 0.000} C_DIS
LIN {X -101.288,Y 7.144,Z -10.363,A 90.000,B 90.000,C 0.000} C_DIS
LIN {X -102.139,Y 7.144,Z -10.784,A 90.000,B 90.000,C 0.000} C_DIS
LIN {X -102.966,Y 7.144,Z -11.251,A 90.000,B 90.000,C 0.000} C_DIS
LIN {X -103.768,Y 7.144,Z -11.761,A 90.000,B 90.000,C 0.000} C_DIS
LIN {X -104.541,Y 7.144,Z -12.312,A 90.000,B 90.000,C 0.000} C_DIS
LIN {X -105.283,Y 7.144,Z -12.905,A 90.000,B 90.000,C 0.000} C_DIS
LIN {X -106.193,Y 7.144,Z -13.027,A 90.000,B 90.000,C 0.000} C_DIS
LIN {X -107.097,Y 7.144,Z -13.184,A 90.000,B 90.000,C 0.000} C_DIS
LIN {X -107.995,Y 7.144,Z -13.374,A 90.000,B 90.000,C 0.000} C_DIS
LIN {X -109.083,Y 7.144,Z -13.619,A 90.000,B 90.000,C 0.000} C_DIS
LIN {X -110.154,Y 7.144,Z -13.929,A 90.000,B 90.000,C 0.000} C_DIS
LIN {X -111.204,Y 7.144,Z -14.303,A 90.000,B 90.000,C 0.000} C_DIS
LIN {X -112.230,Y 7.144,Z -14.740,A 90.000,B 90.000,C 0.000} C_DIS
LIN {X -113.228,Y 7.144,Z -15.237,A 90.000,B 90.000,C 0.000} C_DIS
LIN {X -114.194,Y 7.144,Z -15.794,A 90.000,B 90.000,C 0.000} C_DIS
LIN {X -115.124,Y 7.144,Z -16.408,A 90.000,B 90.000,C 0.000} C_DIS
LIN {X -116.016,Y 7.144,Z -17.077,A 90.000,B 90.000,C 0.000} C_DIS
LIN {X -116.867,Y 7.144,Z -17.799,A 90.000,B 90.000,C 0.000} C_DIS
LIN {X -117.672,Y 7.144,Z -18.570,A 90.000,B 90.000,C 0.000} C_DIS
LIN {X -118.429,Y 7.144,Z -19.389,A 90.000,B 90.000,C 0.000} C_DIS
LIN {X -119.135,Y 7.144,Z -20.252,A 90.000,B 90.000,C 0.000} C_DIS
LIN {X -119.788,Y 7.144,Z -21.155,A 90.000,B 90.000,C 0.000} C_DIS
LIN {X -120.386,Y 7.144,Z -22.097,A 90.000,B 90.000,C 0.000} C_DIS
LIN {X -120.926,Y 7.144,Z -23.072,A 90.000,B 90.000,C 0.000} C_DIS
LIN {X -121.477,Y 7.144,Z -23.671,A 90.000,B 90.000,C 0.000} C_DIS
LIN {X -121.992,Y 7.144,Z -24.302,A 90.000,B 90.000,C 0.000} C_DIS
LIN {X -122.467,Y 7.144,Z -24.963,A 90.000,B 90.000,C 0.000} C_DIS
LIN {X -122.901,Y 7.144,Z -25.652,A 90.000,B 90.000,C 0.000} C_DIS
LIN {X -123.423,Y 7.144,Z -26.483,A 90.000,B 90.000,C 0.000} C_DIS
LIN {X -123.890,Y 7.144,Z -27.346,A 90.000,B 90.000,C 0.000} C_DIS
LIN {X -124.299,Y 7.144,Z -28.239,A 90.000,B 90.000,C 0.000} C_DIS
LIN {X -124.648,Y 7.144,Z -29.156,A 90.000,B 90.000,C 0.000} C_DIS
LIN {X -124.936,Y 7.144,Z -30.094,A 90.000,B 90.000,C 0.000} C_DIS
LIN {X -125.161,Y 7.144,Z -31.049,A 90.000,B 90.000,C 0.000} C_DIS
LIN {X -125.323,Y 7.144,Z -32.017,A 90.000,B 90.000,C 0.000} C_DIS
LIN {X -125.421,Y 7.144,Z -32.994,A 90.000,B 90.000,C 0.000} C_DIS
LIN {X -125.454,Y 7.144,Z -33.975,A 90.000,B 90.000,C 0.000} C_DIS
LIN {X -125.423,Y 7.144,Z -34.956,A 90.000,B 90.000,C 0.000} C_DIS
LIN {X -125.327,Y 7.144,Z -35.933,A 90.000,B 90.000,C 0.000} C_DIS
LIN {X -125.168,Y 7.144,Z -36.901,A 90.000,B 90.000,C 0.000} C_DIS
LIN {X -125.427,Y 7.144,Z -37.908,A 90.000,B 90.000,C 0.000} C_DIS
LIN {X -125.622,Y 7.144,Z -38.929,A 90.000,B 90.000,C 0.000} C_DIS
LIN {X -125.751,Y 7.144,Z -39.960,A 90.000,B 90.000,C 0.000} C_DIS
LIN {X -125.813,Y 7.144,Z -40.998,A 90.000,B 90.000,C 0.000} C_DIS
LIN {X -125.810,Y 7.144,Z -42.037,A 90.000,B 90.000,C 0.000} C_DIS
LIN {X -125.739,Y 7.144,Z -43.074,A 90.000,B 90.000,C 0.000} C_DIS
LIN {X -125.603,Y 7.144,Z -44.105,A 90.000,B 90.000,C 0.000} C_DIS
LIN {X -125.401,Y 7.144,Z -45.124,A 90.000,B 90.000,C 0.000} C_DIS
LIN {X -125.134,Y 7.144,Z -46.129,A 90.000,B 90.000,C 0.000} C_DIS
LIN {X -125.146,Y 7.144,Z -46.198,A 90.000,B 90.000,C 0.000} C_DIS
LIN {X -125.246,Y 7.144,Z -47.329,A 90.000,B 90.000,C 0.000} C_DIS
LIN {X -125.281,Y 7.144,Z -48.464,A 90.000,B 90.000,C 0.000} C_DIS
LIN {X -125.252,Y 7.144,Z -49.599,A 90.000,B 90.000,C 0.000} C_DIS
LIN {X -125.158,Y 7.144,Z -50.731,A 90.000,B 90.000,C 0.000} C_DIS
LIN {X -125.000,Y 7.144,Z -51.855,A 90.000,B 90.000,C 0.000} C_DIS
LIN {X -124.477,Y 7.144,Z -53.720,A 90.000,B 90.000,C 0.000} C_DIS
LIN {X -123.895,Y 7.144,Z -55.567,A 90.000,B 90.000,C 0.000} C_DIS
LIN {X -123.256,Y 7.144,Z -57.395,A 90.000,B 90.000,C 0.000} C_DIS
LIN {X -122.560,Y 7.144,Z -59.202,A 90.000,B 90.000,C 0.000} C_DIS
LIN {X -121.995,Y 7.144,Z -60.983,A 90.000,B 90.000,C 0.000} C_DIS
LIN {X -121.391,Y 7.144,Z -62.751,A 90.000,B 90.000,C 0.000} C_DIS
LIN {X -120.751,Y 7.144,Z -64.506,A 90.000,B 90.000,C 0.000} C_DIS
LIN {X -120.073,Y 7.144,Z -66.248,A 90.000,B 90.000,C 0.000} C_DIS
LIN {X -119.358,Y 7.144,Z -67.974,A 90.000,B 90.000,C 0.000} C_DIS
LIN {X -118.697,Y 7.144,Z -69.282,A 90.000,B 90.000,C 0.000} C_DIS
LIN {X -117.974,Y 7.144,Z -70.556,A 90.000,B 90.000,C 0.000} C_DIS
LIN {X -117.192,Y 7.144,Z -71.795,A 90.000,B 90.000,C 0.000} C_DIS
LIN {X -116.351,Y 7.144,Z -72.996,A 90.000,B 90.000,C 0.000} C_DIS
LIN {X -115.455,Y 7.144,Z -74.154,A 90.000,B 90.000,C 0.000} C_DIS
LIN {X -114.504,Y 7.144,Z -75.269,A 90.000,B 90.000,C 0.000} C_DIS
LIN {X -113.501,Y 7.144,Z -76.338,A 90.000,B 90.000,C 0.000} C_DIS
LIN {X -112.449,Y 7.144,Z -77.357,A 90.000,B 90.000,C 0.000} C_DIS
LIN {X -111.349,Y 7.144,Z -78.325,A 90.000,B 90.000,C 0.000} C_DIS
LIN {X -110.204,Y 7.144,Z -79.240,A 90.000,B 90.000,C 0.000} C_DIS
LIN {X -109.281,Y 7.144,Z -79.997,A 90.000,B 90.000,C 0.000} C_DIS
LIN {X -108.320,Y 7.144,Z -80.705,A 90.000,B 90.000,C 0.000} C_DIS
LIN {X -107.323,Y 7.144,Z -81.362,A 90.000,B 90.000,C 0.000} C_DIS
LIN {X -106.295,Y 7.144,Z -81.967,A 90.000,B 90.000,C 0.000} C_DIS
LIN {X -105.236,Y 7.144,Z -82.519,A 90.000,B 90.000,C 0.000} C_DIS
LIN {X -104.150,Y 7.144,Z -83.015,A 90.000,B 90.000,C 0.000} C_DIS
LIN {X -103.040,Y 7.144,Z -83.454,A 90.000,B 90.000,C 0.000} C_DIS
LIN {X -101.710,Y 7.144,Z -83.860,A 90.000,B 90.000,C 0.000} C_DIS
LIN {X -100.362,Y 7.144,Z -84.202,A 90.000,B 90.000,C 0.000} C_DIS
LIN {X -98.999,Y 7.144,Z -84.479,A 90.000,B 90.000,C 0.000} C_DIS
LIN {X -97.625,Y 7.144,Z -84.691,A 90.000,B 90.000,C 0.000} C_DIS
LIN {X -96.242,Y 7.144,Z -84.836,A 90.000,B 90.000,C 0.000} C_DIS
LIN {X -94.854,Y 7.144,Z -84.916,A 90.000,B 90.000,C 0.000} C_DIS
LIN {X -93.464,Y 7.144,Z -84.929,A 90.000,B 90.000,C 0.000} C_DIS
LIN {X -92.074,Y 7.144,Z -84.876,A 90.000,B 90.000,C 0.000} C_DIS
LIN {X -90.638,Y 7.144,Z -85.887,A 90.000,B 90.000,C 0.000} C_DIS
LIN {X -89.182,Y 7.144,Z -86.867,A 90.000,B 90.000,C 0.000} C_DIS
LIN {X -87.400,Y 7.144,Z -88.248,A 90.000,B 90.000,C 0.000} C_DIS
LIN {X -85.591,Y 7.144,Z -89.594,A 90.000,B 90.000,C 0.000} C_DIS
LIN {X -83.755,Y 7.144,Z -90.903,A 90.000,B 90.000,C 0.000} C_DIS
LIN {X -81.893,Y 7.144,Z -92.174,A 90.000,B 90.000,C 0.000} C_DIS
LIN {X -80.007,Y 7.144,Z -93.409,A 90.000,B 90.000,C 0.000} C_DIS
LIN {X -78.095,Y 7.144,Z -94.604,A 90.000,B 90.000,C 0.000} C_DIS
LIN {X -76.558,Y 7.144,Z -95.551,A 90.000,B 90.000,C 0.000} C_DIS
LIN {X -75.051,Y 7.144,Z -96.545,A 90.000,B 90.000,C 0.000} C_DIS
LIN {X -73.576,Y 7.144,Z -97.586,A 90.000,B 90.000,C 0.000} C_DIS
LIN {X -72.134,Y 7.144,Z -98.673,A 90.000,B 90.000,C 0.000} C_DIS
LIN {X -70.728,Y 7.144,Z -99.804,A 90.000,B 90.000,C 0.000} C_DIS
LIN {X -69.357,Y 7.144,Z -100.979,A 90.000,B 90.000,C 0.000} C_DIS
LIN {X -68.024,Y 7.144,Z -102.197,A 90.000,B 90.000,C 0.000} C_DIS
LIN {X -65.746,Y 7.144,Z -104.601,A 90.000,B 90.000,C 0.000} C_DIS
LIN {X -63.512,Y 7.144,Z -107.047,A 90.000,B 90.000,C 0.000} C_DIS
LIN {X -61.324,Y 7.144,Z -109.533,A 90.000,B 90.000,C 0.000} C_DIS
LIN {X -59.183,Y 7.144,Z -112.059,A 90.000,B 90.000,C 0.000} C_DIS
LIN {X -57.088,Y 7.144,Z -114.625,A 90.000,B 90.000,C 0.000} C_DIS
LIN {X -55.482,Y 7.144,Z -116.471,A 90.000,B 90.000,C 0.000} C_DIS
LIN {X -53.922,Y 7.144,Z -118.356,A 90.000,B 90.000,C 0.000} C_DIS
LIN {X -52.408,Y 7.144,Z -120.278,A 90.000,B 90.000,C 0.000} C_DIS
LIN {X -50.941,Y 7.144,Z -122.237,A 90.000,B 90.000,C 0.000} C_DIS
LIN {X -49.522,Y 7.144,Z -124.230,A 90.000,B 90.000,C 0.000} C_DIS
LIN {X -48.704,Y 7.144,Z -125.822,A 90.000,B 90.000,C 0.000} C_DIS
LIN {X -47.932,Y 7.144,Z -127.436,A 90.000,B 90.000,C 0.000} C_DIS
LIN {X -47.208,Y 7.144,Z -129.073,A 90.000,B 90.000,C 0.000} C_DIS
LIN {X -46.532,Y 7.144,Z -130.730,A 90.000,B 90.000,C 0.000} C_DIS
LIN {X -45.697,Y 7.144,Z -132.758,A 90.000,B 90.000,C 0.000} C_DIS
LIN {X -44.804,Y 7.144,Z -134.761,A 90.000,B 90.000,C 0.000} C_DIS
LIN {X -43.854,Y 7.144,Z -136.738,A 90.000,B 90.000,C 0.000} C_DIS
LIN {X -42.849,Y 7.144,Z -138.687,A 90.000,B 90.000,C 0.000} C_DIS
LIN {X -41.788,Y 7.144,Z -140.607,A 90.000,B 90.000,C 0.000} C_DIS
LIN {X -40.673,Y 7.144,Z -142.496,A 90.000,B 90.000,C 0.000} C_DIS
LIN {X -39.505,Y 7.144,Z -144.352,A 90.000,B 90.000,C 0.000} C_DIS
LIN {X -38.111,Y 7.144,Z -146.320,A 90.000,B 90.000,C 0.000} C_DIS
LIN {X -36.669,Y 7.144,Z -148.254,A 90.000,B 90.000,C 0.000} C_DIS
LIN {X -35.180,Y 7.144,Z -150.151,A 90.000,B 90.000,C 0.000} C_DIS
LIN {X -33.645,Y 7.144,Z -152.011,A 90.000,B 90.000,C 0.000} C_DIS
LIN {X -32.064,Y 7.144,Z -153.833,A 90.000,B 90.000,C 0.000} C_DIS
LIN {X -30.439,Y 7.144,Z -155.616,A 90.000,B 90.000,C 0.000} C_DIS
LIN {X -28.771,Y 7.144,Z -157.358,A 90.000,B 90.000,C 0.000} C_DIS
LIN {X -26.290,Y 7.144,Z -160.015,A 90.000,B 90.000,C 0.000} C_DIS
LIN {X -25.814,Y 7.144,Z -160.540,A 90.000,B 90.000,C 0.000} C_DIS
LIN {X -25.380,Y 7.144,Z -161.100,A 90.000,B 90.000,C 0.000} C_DIS
LIN {X -24.988,Y 7.144,Z -161.690,A 90.000,B 90.000,C 0.000} C_DIS
LIN {X -24.643,Y 7.144,Z -162.309,A 90.000,B 90.000,C 0.000} C_DIS
LIN {X -25.107,Y 7.144,Z -163.539,A 90.000,B 90.000,C 0.000} C_DIS
LIN {X -25.634,Y 7.144,Z -164.743,A 90.000,B 90.000,C 0.000} C_DIS
LIN {X -26.223,Y 7.144,Z -165.918,A 90.000,B 90.000,C 0.000} C_DIS
LIN {X -26.871,Y 7.144,Z -167.062,A 90.000,B 90.000,C 0.000} C_DIS
LIN {X -27.577,Y 7.144,Z -168.170,A 90.000,B 90.000,C 0.000} C_DIS
LIN {X -28.340,Y 7.144,Z -169.241,A 90.000,B 90.000,C 0.000} C_DIS
LIN {X -29.156,Y 7.144,Z -170.271,A 90.000,B 90.000,C 0.000} C_DIS
LIN {X -30.662,Y 7.144,Z -171.784,A 90.000,B 90.000,C 0.000} C_DIS
LIN {X -32.211,Y 7.144,Z -173.253,A 90.000,B 90.000,C 0.000} C_DIS
LIN {X -33.803,Y 7.144,Z -174.675,A 90.000,B 90.000,C 0.000} C_DIS
LIN {X -35.436,Y 7.144,Z -176.050,A 90.000,B 90.000,C 0.000} C_DIS
LIN {X -37.109,Y 7.144,Z -177.376,A 90.000,B 90.000,C 0.000} C_DIS
LIN {X -38.820,Y 7.144,Z -178.653,A 90.000,B 90.000,C 0.000} C_DIS
LIN {X -42.083,Y 7.144,Z -180.979,A 90.000,B 90.000,C 0.000} C_DIS
LIN {X -45.382,Y 7.144,Z -183.254,A 90.000,B 90.000,C 0.000} C_DIS
LIN {X -48.716,Y 7.144,Z -185.478,A 90.000,B 90.000,C 0.000} C_DIS
LIN {X -52.083,Y 7.144,Z -187.651,A 90.000,B 90.000,C 0.000} C_DIS
LIN {X -55.483,Y 7.144,Z -189.771,A 90.000,B 90.000,C 0.000} C_DIS
LIN {X -58.916,Y 7.144,Z -191.839,A 90.000,B 90.000,C 0.000} C_DIS
LIN {X -62.380,Y 7.144,Z -193.854,A 90.000,B 90.000,C 0.000} C_DIS
LIN {X -65.874,Y 7.144,Z -195.816,A 90.000,B 90.000,C 0.000} C_DIS
LIN {X -71.584,Y 7.144,Z -198.984,A 90.000,B 90.000,C 0.000} C_DIS
LIN {X -77.266,Y 7.144,Z -202.204,A 90.000,B 90.000,C 0.000} C_DIS
LIN {X -82.919,Y 7.144,Z -205.474,A 90.000,B 90.000,C 0.000} C_DIS
LIN {X -88.542,Y 7.144,Z -208.795,A 90.000,B 90.000,C 0.000} C_DIS
LIN {X -94.136,Y 7.144,Z -212.166,A 90.000,B 90.000,C 0.000} C_DIS
LIN {X -99.699,Y 7.144,Z -215.587,A 90.000,B 90.000,C 0.000} C_DIS
LIN {X -105.231,Y 7.144,Z -219.057,A 90.000,B 90.000,C 0.000} C_DIS
LIN {X -110.731,Y 7.144,Z -222.577,A 90.000,B 90.000,C 0.000} C_DIS
LIN {X -116.200,Y 7.144,Z -226.147,A 90.000,B 90.000,C 0.000} C_DIS
LIN {X -130.828,Y 7.144,Z -235.748,A 90.000,B 90.000,C 0.000} C_DIS
LIN {X -137.589,Y 7.144,Z -240.214,A 90.000,B 90.000,C 0.000} C_DIS
LIN {X -138.176,Y 7.144,Z -240.685,A 90.000,B 90.000,C 0.000} C_DIS
LIN {X -138.730,Y 7.144,Z -241.194,A 90.000,B 90.000,C 0.000} C_DIS
LIN {X -139.249,Y 7.144,Z -241.739,A 90.000,B 90.000,C 0.000} C_DIS
LIN {X -139.731,Y 7.144,Z -242.317,A 90.000,B 90.000,C 0.000} C_DIS
LIN {X -140.174,Y 7.144,Z -242.925,A 90.000,B 90.000,C 0.000} C_DIS
LIN {X -140.576,Y 7.144,Z -243.561,A 90.000,B 90.000,C 0.000} C_DIS
LIN {X -145.015,Y 7.144,Z -243.561,A 90.000,B 90.000,C 0.000} C_DIS
LIN {X -145.015,Y 7.144,Z 0.000,A 90.000,B 90.000,C 0.000} C_DIS
LIN {X 145.015,Y 7.144,Z 0.000,A 90.000,B 90.000,C 0.000} C_DIS
LIN {X 145.015,Y 7.144,Z -243.561,A 90.000,B 90.000,C 0.000} C_DIS
LIN {X 104.284,Y 7.144,Z -243.561,A 90.000,B 90.000,C 0.000} C_DIS
LIN {X 105.298,Y 7.144,Z -240.765,A 90.000,B 90.000,C 0.000} C_DIS
LIN {X 106.267,Y 7.144,Z -237.954,A 90.000,B 90.000,C 0.000} C_DIS
LIN {X 107.192,Y 7.144,Z -235.128,A 90.000,B 90.000,C 0.000} C_DIS
LIN {X 108.072,Y 7.144,Z -232.287,A 90.000,B 90.000,C 0.000} C_DIS
LIN {X 108.907,Y 7.144,Z -229.433,A 90.000,B 90.000,C 0.000} C_DIS
LIN {X 109.697,Y 7.144,Z -226.566,A 90.000,B 90.000,C 0.000} C_DIS
LIN {X 110.662,Y 7.144,Z -222.495,A 90.000,B 90.000,C 0.000} C_DIS
LIN {X 111.574,Y 7.144,Z -218.413,A 90.000,B 90.000,C 0.000} C_DIS
LIN {X 112.432,Y 7.144,Z -214.318,A 90.000,B 90.000,C 0.000} C_DIS
LIN {X 113.236,Y 7.144,Z -210.213,A 90.000,B 90.000,C 0.000} C_DIS
LIN {X 113.987,Y 7.144,Z -206.097,A 90.000,B 90.000,C 0.000} C_DIS
LIN {X 114.684,Y 7.144,Z -201.972,A 90.000,B 90.000,C 0.000} C_DIS
LIN {X 115.327,Y 7.144,Z -197.839,A 90.000,B 90.000,C 0.000} C_DIS
LIN {X 115.916,Y 7.144,Z -193.697,A 90.000,B 90.000,C 0.000} C_DIS
LIN {X 116.548,Y 7.144,Z -188.440,A 90.000,B 90.000,C 0.000} C_DIS
LIN {X 117.125,Y 7.144,Z -183.178,A 90.000,B 90.000,C 0.000} C_DIS
LIN {X 117.648,Y 7.144,Z -177.909,A 90.000,B 90.000,C 0.000} C_DIS
LIN {X 118.116,Y 7.144,Z -172.635,A 90.000,B 90.000,C 0.000} C_DIS
LIN {X 118.530,Y 7.144,Z -167.357,A 90.000,B 90.000,C 0.000} C_DIS
LIN {X 118.889,Y 7.144,Z -162.075,A 90.000,B 90.000,C 0.000} C_DIS
LIN {X 119.193,Y 7.144,Z -156.789,A 90.000,B 90.000,C 0.000} C_DIS
LIN {X 119.407,Y 7.144,Z -153.299,A 90.000,B 90.000,C 0.000} C_DIS
LIN {X 119.553,Y 7.144,Z -149.806,A 90.000,B 90.000,C 0.000} C_DIS
LIN {X 119.633,Y 7.144,Z -146.311,A 90.000,B 90.000,C 0.000} C_DIS
LIN {X 119.645,Y 7.144,Z -142.815,A 90.000,B 90.000,C 0.000} C_DIS
LIN {X 119.590,Y 7.144,Z -139.319,A 90.000,B 90.000,C 0.000} C_DIS
LIN {X 119.469,Y 7.144,Z -135.825,A 90.000,B 90.000,C 0.000} C_DIS
LIN {X 119.280,Y 7.144,Z -132.334,A 90.000,B 90.000,C 0.000} C_DIS
LIN {X 119.025,Y 7.144,Z -128.847,A 90.000,B 90.000,C 0.000} C_DIS
LIN {X 118.596,Y 7.144,Z -124.844,A 90.000,B 90.000,C 0.000} C_DIS
LIN {X 118.099,Y 7.144,Z -120.848,A 90.000,B 90.000,C 0.000} C_DIS
LIN {X 117.534,Y 7.144,Z -116.862,A 90.000,B 90.000,C 0.000} C_DIS
LIN {X 116.901,Y 7.144,Z -112.886,A 90.000,B 90.000,C 0.000} C_DIS
LIN {X 116.200,Y 7.144,Z -108.921,A 90.000,B 90.000,C 0.000} C_DIS
LIN {X 115.431,Y 7.144,Z -104.969,A 90.000,B 90.000,C 0.000} C_DIS
LIN {X 114.595,Y 7.144,Z -101.030,A 90.000,B 90.000,C 0.000} C_DIS
LIN {X 113.692,Y 7.144,Z -97.107,A 90.000,B 90.000,C 0.000} C_DIS
LIN {X 112.722,Y 7.144,Z -93.199,A 90.000,B 90.000,C 0.000} C_DIS
LIN {X 112.268,Y 7.144,Z -91.576,A 90.000,B 90.000,C 0.000} C_DIS
LIN {X 111.753,Y 7.144,Z -89.970,A 90.000,B 90.000,C 0.000} C_DIS
LIN {X 111.179,Y 7.144,Z -88.385,A 90.000,B 90.000,C 0.000} C_DIS
LIN {X 110.547,Y 7.144,Z -86.822,A 90.000,B 90.000,C 0.000} C_DIS
LIN {X 109.858,Y 7.144,Z -85.283,A 90.000,B 90.000,C 0.000} C_DIS
LIN {X 109.111,Y 7.144,Z -83.772,A 90.000,B 90.000,C 0.000} C_DIS
LIN {X 110.148,Y 7.144,Z -81.952,A 90.000,B 90.000,C 0.000} C_DIS
LIN {X 111.135,Y 7.144,Z -80.105,A 90.000,B 90.000,C 0.000} C_DIS
LIN {X 112.071,Y 7.144,Z -78.232,A 90.000,B 90.000,C 0.000} C_DIS
LIN {X 112.956,Y 7.144,Z -76.334,A 90.000,B 90.000,C 0.000} C_DIS
LIN {X 113.790,Y 7.144,Z -74.413,A 90.000,B 90.000,C 0.000} C_DIS
LIN {X 114.571,Y 7.144,Z -72.470,A 90.000,B 90.000,C 0.000} C_DIS
LIN {X 115.299,Y 7.144,Z -70.506,A 90.000,B 90.000,C 0.000} C_DIS
LIN {X 115.973,Y 7.144,Z -68.523,A 90.000,B 90.000,C 0.000} C_DIS
LIN {X 116.594,Y 7.144,Z -66.523,A 90.000,B 90.000,C 0.000} C_DIS
LIN {X 117.391,Y 7.144,Z -63.629,A 90.000,B 90.000,C 0.000} C_DIS
LIN {X 118.216,Y 7.144,Z -60.743,A 90.000,B 90.000,C 0.000} C_DIS
LIN {X 118.900,Y 7.144,Z -58.947,A 90.000,B 90.000,C 0.000} C_DIS
LIN {X 119.632,Y 7.144,Z -57.170,A 90.000,B 90.000,C 0.000} C_DIS
LIN {X 120.411,Y 7.144,Z -55.413,A 90.000,B 90.000,C 0.000} C_DIS
LIN {X 121.238,Y 7.144,Z -53.679,A 90.000,B 90.000,C 0.000} C_DIS
LIN {X 122.112,Y 7.144,Z -51.967,A 90.000,B 90.000,C 0.000} C_DIS
LIN {X 122.620,Y 7.144,Z -50.961,A 90.000,B 90.000,C 0.000} C_DIS
LIN {X 123.069,Y 7.144,Z -49.926,A 90.000,B 90.000,C 0.000} C_DIS
LIN {X 123.455,Y 7.144,Z -48.867,A 90.000,B 90.000,C 0.000} C_DIS
LIN {X 123.778,Y 7.144,Z -47.788,A 90.000,B 90.000,C 0.000} C_DIS
LIN {X 124.038,Y 7.144,Z -46.690,A 90.000,B 90.000,C 0.000} C_DIS
LIN {X 124.232,Y 7.144,Z -45.580,A 90.000,B 90.000,C 0.000} C_DIS
LIN {X 124.360,Y 7.144,Z -44.460,A 90.000,B 90.000,C 0.000} C_DIS
LIN {X 124.422,Y 7.144,Z -43.334,A 90.000,B 90.000,C 0.000} C_DIS
LIN {X 124.417,Y 7.144,Z -42.207,A 90.000,B 90.000,C 0.000} C_DIS
LIN {X 124.347,Y 7.144,Z -41.082,A 90.000,B 90.000,C 0.000} C_DIS
LIN {X 124.254,Y 7.144,Z -40.095,A 90.000,B 90.000,C 0.000} C_DIS
LIN {X 124.088,Y 7.144,Z -39.117,A 90.000,B 90.000,C 0.000} C_DIS
LIN {X 123.849,Y 7.144,Z -38.155,A 90.000,B 90.000,C 0.000} C_DIS
LIN {X 123.540,Y 7.144,Z -37.213,A 90.000,B 90.000,C 0.000} C_DIS
LIN {X 123.161,Y 7.144,Z -36.296,A 90.000,B 90.000,C 0.000} C_DIS
LIN {X 122.715,Y 7.144,Z -35.411,A 90.000,B 90.000,C 0.000} C_DIS
LIN {X 122.205,Y 7.144,Z -34.561,A 90.000,B 90.000,C 0.000} C_DIS
LIN {X 121.633,Y 7.144,Z -33.751,A 90.000,B 90.000,C 0.000} C_DIS
LIN {X 121.002,Y 7.144,Z -32.986,A 90.000,B 90.000,C 0.000} C_DIS
LIN {X 120.316,Y 7.144,Z -32.270,A 90.000,B 90.000,C 0.000} C_DIS
LIN {X 119.578,Y 7.144,Z -31.607,A 90.000,B 90.000,C 0.000} C_DIS
LIN {X 118.794,Y 7.144,Z -31.001,A 90.000,B 90.000,C 0.000} C_DIS
LIN {X 117.966,Y 7.144,Z -30.455,A 90.000,B 90.000,C 0.000} C_DIS
LIN {X 117.834,Y 7.144,Z -30.373,A 90.000,B 90.000,C 0.000} C_DIS
LIN {X 116.952,Y 7.144,Z -29.886,A 90.000,B 90.000,C 0.000} C_DIS
LIN {X 116.037,Y 7.144,Z -29.462,A 90.000,B 90.000,C 0.000} C_DIS
LIN {X 115.095,Y 7.144,Z -29.104,A 90.000,B 90.000,C 0.000} C_DIS
LIN {X 114.129,Y 7.144,Z -28.814,A 90.000,B 90.000,C 0.000} C_DIS
LIN {X 113.146,Y 7.144,Z -28.594,A 90.000,B 90.000,C 0.000} C_DIS
LIN {X 112.149,Y 7.144,Z -28.443,A 90.000,B 90.000,C 0.000} C_DIS
LIN {X 111.144,Y 7.144,Z -28.364,A 90.000,B 90.000,C 0.000} C_DIS
LIN {X 110.136,Y 7.144,Z -28.356,A 90.000,B 90.000,C 0.000} C_DIS
LIN {X 109.131,Y 7.144,Z -28.420,A 90.000,B 90.000,C 0.000} C_DIS
LIN {X 108.132,Y 7.144,Z -28.555,A 90.000,B 90.000,C 0.000} C_DIS
LIN {X 107.145,Y 7.144,Z -28.761,A 90.000,B 90.000,C 0.000} C_DIS
LIN {X 105.492,Y 7.144,Z -29.303,A 90.000,B 90.000,C 0.000} C_DIS
LIN {X 103.857,Y 7.144,Z -29.898,A 90.000,B 90.000,C 0.000} C_DIS
LIN {X 102.242,Y 7.144,Z -30.545,A 90.000,B 90.000,C 0.000} C_DIS
LIN {X 100.649,Y 7.144,Z -31.243,A 90.000,B 90.000,C 0.000} C_DIS
LIN {X 98.913,Y 7.144,Z -31.951,A 90.000,B 90.000,C 0.000} C_DIS
LIN {X 97.202,Y 7.144,Z -32.718,A 90.000,B 90.000,C 0.000} C_DIS
LIN {X 95.519,Y 7.144,Z -33.544,A 90.000,B 90.000,C 0.000} C_DIS
LIN {X 93.866,Y 7.144,Z -34.428,A 90.000,B 90.000,C 0.000} C_DIS
LIN {X 92.244,Y 7.144,Z -35.368,A 90.000,B 90.000,C 0.000} C_DIS
LIN {X 90.655,Y 7.144,Z -36.364,A 90.000,B 90.000,C 0.000} C_DIS
LIN {X 89.102,Y 7.144,Z -37.414,A 90.000,B 90.000,C 0.000} C_DIS
LIN {X 87.585,Y 7.144,Z -38.517,A 90.000,B 90.000,C 0.000} C_DIS
LIN {X 86.108,Y 7.144,Z -39.671,A 90.000,B 90.000,C 0.000} C_DIS
LIN {X 84.940,Y 7.144,Z -40.598,A 90.000,B 90.000,C 0.000} C_DIS
LIN {X 83.816,Y 7.144,Z -41.577,A 90.000,B 90.000,C 0.000} C_DIS
LIN {X 82.738,Y 7.144,Z -42.607,A 90.000,B 90.000,C 0.000} C_DIS
LIN {X 81.708,Y 7.144,Z -43.685,A 90.000,B 90.000,C 0.000} C_DIS
LIN {X 80.729,Y 7.144,Z -44.810,A 90.000,B 90.000,C 0.000} C_DIS
LIN {X 79.803,Y 7.144,Z -45.978,A 90.000,B 90.000,C 0.000} C_DIS
LIN {X 78.931,Y 7.144,Z -47.188,A 90.000,B 90.000,C 0.000} C_DIS
LIN {X 78.116,Y 7.144,Z -48.436,A 90.000,B 90.000,C 0.000} C_DIS
LIN {X 78.116,Y 19.644,Z -48.436,A 90.000,B 90.000,C 0.000} C_DIS
LIN {X 78.116,Y 32.144,Z -48.436,A 90.000,B 90.000,C 0.000} C_DIS
LIN {X 78.116,Y 58.537,Z -48.436,A 90.000,B 90.000,C 0.000} C_DIS
LIN {X 144.015,Y 58.537,Z -242.561,A 90.000,B 90.000,C 0.000} C_DIS
LIN {X 144.015,Y 25.000,Z -242.561,A 90.000,B 90.000,C 0.000} C_DIS
LIN {X 144.015,Y 12.500,Z -242.561,A 90.000,B 90.000,C 0.000} C_DIS
LIN {X 144.015,Y 0.000,Z -242.561,A 90.000,B 90.000,C 0.000} C_DIS
LIN {X 132.537,Y 0.000,Z -242.561,A 90.000,B 90.000,C 0.000} C_DIS
LIN {X 132.537,Y 0.000,Z -235.012,A 90.000,B 90.000,C 0.000} C_DIS
LIN {X 144.015,Y 0.000,Z -235.012,A 90.000,B 90.000,C 0.000} C_DIS
LIN {X 144.015,Y 0.000,Z -227.464,A 90.000,B 90.000,C 0.000} C_DIS
LIN {X 132.537,Y 0.000,Z -227.464,A 90.000,B 90.000,C 0.000} C_DIS
LIN {X 132.537,Y 0.000,Z -219.915,A 90.000,B 90.000,C 0.000} C_DIS
LIN {X 144.015,Y 0.000,Z -219.915,A 90.000,B 90.000,C 0.000} C_DIS
LIN {X 144.015,Y 0.000,Z -212.366,A 90.000,B 90.000,C 0.000} C_DIS
LIN {X 132.537,Y 0.000,Z -212.366,A 90.000,B 90.000,C 0.000} C_DIS
LIN {X 132.537,Y 0.000,Z -204.817,A 90.000,B 90.000,C 0.000} C_DIS
LIN {X 144.015,Y 0.000,Z -204.817,A 90.000,B 90.000,C 0.000} C_DIS
LIN {X 144.015,Y 0.000,Z -197.269,A 90.000,B 90.000,C 0.000} C_DIS
LIN {X 132.537,Y 0.000,Z -197.269,A 90.000,B 90.000,C 0.000} C_DIS
LIN {X 132.537,Y 0.000,Z -189.720,A 90.000,B 90.000,C 0.000} C_DIS
LIN {X 144.015,Y 0.000,Z -189.720,A 90.000,B 90.000,C 0.000} C_DIS
LIN {X 144.015,Y 0.000,Z -182.171,A 90.000,B 90.000,C 0.000} C_DIS
LIN {X 132.537,Y 0.000,Z -182.171,A 90.000,B 90.000,C 0.000} C_DIS
LIN {X 132.537,Y 0.000,Z -174.622,A 90.000,B 90.000,C 0.000} C_DIS
LIN {X 144.015,Y 0.000,Z -174.622,A 90.000,B 90.000,C 0.000} C_DIS
LIN {X 144.015,Y 0.000,Z -167.073,A 90.000,B 90.000,C 0.000} C_DIS
LIN {X 132.537,Y 0.000,Z -167.073,A 90.000,B 90.000,C 0.000} C_DIS
LIN {X 132.537,Y 0.000,Z -159.525,A 90.000,B 90.000,C 0.000} C_DIS
LIN {X 144.015,Y 0.000,Z -159.525,A 90.000,B 90.000,C 0.000} C_DIS
LIN {X 144.015,Y 0.000,Z -151.976,A 90.000,B 90.000,C 0.000} C_DIS
LIN {X 132.537,Y 0.000,Z -151.976,A 90.000,B 90.000,C 0.000} C_DIS
LIN {X 132.537,Y 0.000,Z -144.427,A 90.000,B 90.000,C 0.000} C_DIS
LIN {X 144.015,Y 0.000,Z -144.427,A 90.000,B 90.000,C 0.000} C_DIS
LIN {X 144.015,Y 0.000,Z -136.878,A 90.000,B 90.000,C 0.000} C_DIS
LIN {X 132.537,Y 0.000,Z -136.878,A 90.000,B 90.000,C 0.000} C_DIS
LIN {X 132.537,Y 0.000,Z -129.329,A 90.000,B 90.000,C 0.000} C_DIS
LIN {X 144.015,Y 0.000,Z -129.329,A 90.000,B 90.000,C 0.000} C_DIS
LIN {X 144.015,Y 0.000,Z -121.781,A 90.000,B 90.000,C 0.000} C_DIS
LIN {X 132.537,Y 0.000,Z -121.781,A 90.000,B 90.000,C 0.000} C_DIS
LIN {X 132.537,Y 0.000,Z -114.232,A 90.000,B 90.000,C 0.000} C_DIS
LIN {X 144.015,Y 0.000,Z -114.232,A 90.000,B 90.000,C 0.000} C_DIS
LIN {X 144.015,Y 0.000,Z -106.683,A 90.000,B 90.000,C 0.000} C_DIS
LIN {X 132.537,Y 0.000,Z -106.683,A 90.000,B 90.000,C 0.000} C_DIS
LIN {X 132.537,Y 0.000,Z -99.134,A 90.000,B 90.000,C 0.000} C_DIS
LIN {X 144.015,Y 0.000,Z -99.134,A 90.000,B 90.000,C 0.000} C_DIS
LIN {X 144.015,Y 0.000,Z -91.586,A 90.000,B 90.000,C 0.000} C_DIS
LIN {X 132.537,Y 0.000,Z -91.586,A 90.000,B 90.000,C 0.000} C_DIS
LIN {X 132.537,Y 0.000,Z -84.037,A 90.000,B 90.000,C 0.000} C_DIS
LIN {X 144.015,Y 0.000,Z -84.037,A 90.000,B 90.000,C 0.000} C_DIS
LIN {X 144.015,Y 0.000,Z -76.488,A 90.000,B 90.000,C 0.000} C_DIS
LIN {X 132.537,Y 0.000,Z -76.488,A 90.000,B 90.000,C 0.000} C_DIS
LIN {X 132.537,Y 0.000,Z -68.939,A 90.000,B 90.000,C 0.000} C_DIS
LIN {X 144.015,Y 0.000,Z -68.939,A 90.000,B 90.000,C 0.000} C_DIS
LIN {X 144.015,Y 0.000,Z -61.390,A 90.000,B 90.000,C 0.000} C_DIS
LIN {X 132.537,Y 0.000,Z -61.390,A 90.000,B 90.000,C 0.000} C_DIS
LIN {X 132.537,Y 0.000,Z -53.842,A 90.000,B 90.000,C 0.000} C_DIS
LIN {X 144.015,Y 0.000,Z -53.842,A 90.000,B 90.000,C 0.000} C_DIS
LIN {X 144.015,Y 0.000,Z -46.293,A 90.000,B 90.000,C 0.000} C_DIS
LIN {X 132.537,Y 0.000,Z -46.293,A 90.000,B 90.000,C 0.000} C_DIS
LIN {X 132.537,Y 0.000,Z -38.744,A 90.000,B 90.000,C 0.000} C_DIS
LIN {X 144.015,Y 0.000,Z -38.744,A 90.000,B 90.000,C 0.000} C_DIS
LIN {X 144.015,Y 0.000,Z -31.195,A 90.000,B 90.000,C 0.000} C_DIS
LIN {X 132.537,Y 0.000,Z -31.195,A 90.000,B 90.000,C 0.000} C_DIS
LIN {X 132.537,Y 0.000,Z -23.646,A 90.000,B 90.000,C 0.000} C_DIS
LIN {X 144.015,Y 0.000,Z -23.646,A 90.000,B 90.000,C 0.000} C_DIS
LIN {X 144.015,Y 0.000,Z -16.098,A 90.000,B 90.000,C 0.000} C_DIS
LIN {X 132.537,Y 0.000,Z -16.098,A 90.000,B 90.000,C 0.000} C_DIS
LIN {X 132.537,Y 0.000,Z -8.549,A 90.000,B 90.000,C 0.000} C_DIS
LIN {X 144.015,Y 0.000,Z -8.549,A 90.000,B 90.000,C 0.000} C_DIS
LIN {X 144.015,Y 0.000,Z -1.000,A 90.000,B 90.000,C 0.000} C_DIS
LIN {X 132.537,Y 0.000,Z -1.000,A 90.000,B 90.000,C 0.000} C_DIS
LIN {X 131.537,Y 0.000,Z -0.237,A 90.000,B 90.000,C 0.000} C_DIS
LIN {X 131.527,Y 0.000,Z 0.000,A 90.000,B 90.000,C 0.000} C_DIS
LIN {X 145.015,Y 0.000,Z 0.000,A 90.000,B 90.000,C 0.000} C_DIS
LIN {X 145.015,Y 0.000,Z -243.561,A 90.000,B 90.000,C 0.000} C_DIS
LIN {X 131.537,Y 0.000,Z -243.561,A 90.000,B 90.000,C 0.000} C_DIS
LIN {X 131.537,Y 0.000,Z -0.237,A 90.000,B 90.000,C 0.000} C_DIS
LIN {X 131.537,Y 12.500,Z -0.237,A 90.000,B 90.000,C 0.000} C_DIS
LIN {X 131.537,Y 75.000,Z -0.237,A 90.000,B 90.000,C 0.000} C_DIS
LIN {X -141.869,Y 75.000,Z -242.561,A 90.000,B 90.000,C 0.000} C_DIS
LIN {X -141.869,Y 12.500,Z -242.561,A 90.000,B 90.000,C 0.000} C_DIS
